  Set speed (1000.0 mm/s)
  MoveL 10131 to (504.54, 495.95, 18.9) mm, rotated rx 0 ry 90 rz 0 deg; joints [-11.552, -28.213, 111.281, -15.587, -82.457, 51.087]
  Set speed (1000.0 mm/s)
  MoveL 10132 to (501.11, 498.89, 18.9) mm, rotated rx 0 ry 90 rz 0 deg; joints [-11.886, -28.268, 111.619, -15.914, -82.741, 51.048]
  Set speed (30.0 mm/s)
  Call Extruder(0.111)
  MoveL 10133 to (503.8, 496.2, 18.9) mm, rotated rx 0 ry 90 rz 0 deg; joints [-11.588, -28.227, 111.363, -15.622, -82.525, 51.072]
  MoveL 10134 to (503.92, 496.08, 18.9) mm, rotated rx 0 ry 90 rz 0 deg; joints [-11.575, -28.225, 111.352, -15.608, -82.515, 51.073]
  Set speed (120.0 mm/s)
  MoveL 10135 to (504.54, 493.58, 18.9) mm, rotated rx 0 ry 90 rz 0 deg; joints [-11.335, -28.223, 111.338, -15.367, -82.497, 51.049]
  Set speed (1000.0 mm/s)
  MoveL 10136 to (495.89, 493.58, 18.9) mm, rotated rx 0 ry 90 rz 0 deg; joints [-11.496, -28.386, 112.372, -15.5, -83.341, 50.833]
  Set speed (1000.0 mm/s)
  MoveL 10137 to (498.94, 501.06, 18.9) mm, rotated rx 0 ry 90 rz 0 deg; joints [-12.126, -28.301, 111.823, -16.15, -82.913, 51.027]
  Set speed (30.0 mm/s)
  Call Extruder(0.126)
  MoveL 10138 to (495.87, 504.12, 18.9) mm, rotated rx 0 ry 90 rz 0 deg; joints [-12.469, -28.346, 112.108, -16.487, -83.155, 50.995]
  MoveL 10139 to (495.75, 504.25, 18.9) mm, rotated rx 0 ry 90 rz 0 deg; joints [-12.483, -28.347, 112.12, -16.501, -83.165, 50.994]
  Set speed (120.0 mm/s)
  MoveL 10140 to (495.98, 506.75, 18.9) mm, rotated rx 0 ry 90 rz 0 deg; joints [-12.708, -28.333, 112.027, -16.73, -83.096, 51.04]
  Set speed (1000.0 mm/s)
  MoveL 10141 to (504.36, 506.75, 18.9) mm, rotated rx 0 ry 90 rz 0 deg; joints [-12.537, -28.171, 111.026, -16.588, -82.287, 51.263]
  Set speed (1000.0 mm/s)
  MoveL 10142 to (503.43, 503.43, 18.9) mm, rotated rx 0 ry 90 rz 0 deg; joints [-12.254, -28.204, 111.225, -16.297, -82.436, 51.182]
  Set speed (30.0 mm/s)
  Call Extruder(0.243)
  MoveL 10143 to (509.32, 509.32, 18.9) mm, rotated rx 0 ry 90 rz 0 deg; joints [-12.669, -28.058, 110.36, -16.744, -81.762, 51.44]
  MoveL 10144 to (509.44, 509.44, 18.9) mm, rotated rx 0 ry 90 rz 0 deg; joints [-12.677, -28.055, 110.342, -16.753, -81.748, 51.445]
  Set speed (120.0 mm/s)
  MoveL 10145 to (495.98, 506.75, 18.9) mm, rotated rx 0 ry 90 rz 0 deg; joints [-12.708, -28.333, 112.027, -16.73, -83.096, 51.04]
  Set speed (1000.0 mm/s)
  MoveL 10146 to (495.94, 504.34, 18.9) mm, rotated rx 0 ry 90 rz 0 deg; joints [-12.487, -28.344, 112.096, -16.506, -83.145, 51]
  Set speed (1000.0 mm/s)
  MoveL 10147 to (496.01, 504.4, 18.9) mm, rotated rx 0 ry 90 rz 0 deg; joints [-12.492, -28.342, 112.085, -16.511, -83.137, 51.003]
  Set speed (15.0 mm/s)
  Call Extruder(0.067)
  MoveL 10148 to (496.01, 506.72, 18.9) mm, rotated rx 0 ry 90 rz 0 deg; joints [-12.705, -28.332, 112.024, -16.727, -83.094, 51.04]
  Call Extruder(0.242)
  MoveL 10149 to (504.33, 506.72, 18.9) mm, rotated rx 0 ry 90 rz 0 deg; joints [-12.535, -28.172, 111.03, -16.586, -82.29, 51.262]
  Call Extruder(0.027)
  MoveL 10150 to (504.33, 505.8, 18.9) mm, rotated rx 0 ry 90 rz 0 deg; joints [-12.452, -28.176, 111.055, -16.502, -82.307, 51.246]
  Call Extruder(0.306)
  MoveL 10151 to (499.53, 496.43, 18.9) mm, rotated rx 0 ry 90 rz 0 deg; joints [-11.69, -28.308, 111.869, -15.709, -82.937, 50.968]
  Call Extruder(0.017)
  MoveL 10152 to (499.27, 495.92, 18.9) mm, rotated rx 0 ry 90 rz 0 deg; joints [-11.648, -28.315, 111.913, -15.666, -82.971, 50.954]
  Call Extruder(0.010)
  MoveL 10153 to (499.84, 495.92, 18.9) mm, rotated rx 0 ry 90 rz 0 deg; joints [-11.637, -28.304, 111.844, -15.657, -82.916, 50.968]
  Call Extruder(0.000)
  MoveL 10154 to (499.84, 495.92, 18.9) mm, rotated rx 0 ry 90 rz 0 deg; joints [-11.637, -28.304, 111.844, -15.657, -82.915, 50.968]
  Call Extruder(0.136)
  MoveL 10155 to (504.51, 495.92, 18.9) mm, rotated rx 0 ry 90 rz 0 deg; joints [-11.55, -28.214, 111.285, -15.585, -82.461, 51.086]
  Call Extruder(0.067)
  MoveL 10156 to (504.51, 493.61, 18.9) mm, rotated rx 0 ry 90 rz 0 deg; joints [-11.338, -28.223, 111.341, -15.37, -82.499, 51.048]
  Call Extruder(0.250)
  MoveL 10157 to (495.92, 493.61, 18.9) mm, rotated rx 0 ry 90 rz 0 deg; joints [-11.498, -28.386, 112.368, -15.502, -83.338, 50.834]
  Call Extruder(0.027)
  MoveL 10158 to (495.92, 494.52, 18.9) mm, rotated rx 0 ry 90 rz 0 deg; joints [-11.583, -28.382, 112.346, -15.588, -83.322, 50.847]
  Call Extruder(0.306)
  MoveL 10159 to (500.7, 503.9, 18.9) mm, rotated rx 0 ry 90 rz 0 deg; joints [-12.351, -28.255, 111.539, -16.385, -82.691, 51.119]
  Call Extruder(0.017)
  MoveL 10160 to (500.96, 504.4, 18.9) mm, rotated rx 0 ry 90 rz 0 deg; joints [-12.392, -28.248, 111.494, -16.428, -82.657, 51.134]
  Call Extruder(0.010)
  MoveL 10161 to (500.39, 504.41, 18.9) mm, rotated rx 0 ry 90 rz 0 deg; joints [-12.404, -28.259, 111.562, -16.437, -82.712, 51.119]
  Call Extruder(0.000)
  MoveL 10162 to (500.39, 504.41, 18.9) mm, rotated rx 0 ry 90 rz 0 deg; joints [-12.404, -28.259, 111.563, -16.437, -82.712, 51.119]
  Call Extruder(0.128)
  MoveL 10163 to (496.01, 504.4, 18.9) mm, rotated rx 0 ry 90 rz 0 deg; joints [-12.492, -28.342, 112.085, -16.511, -83.137, 51.003]
  Set speed (120.0 mm/s)
  MoveL 10164 to (496.01, 504.8, 18.9) mm, rotated rx 0 ry 90 rz 0 deg; joints [-12.529, -28.34, 112.075, -16.548, -83.13, 51.01]
  Set speed (1000.0 mm/s)
  MoveL 10165 to (495.91, 504.81, 18.9) mm, rotated rx 0 ry 90 rz 0 deg; joints [-12.531, -28.342, 112.087, -16.55, -83.139, 51.007]
  Set speed (1000.0 mm/s)
  MoveL 10166 to (490.47, 509.53, 18.9) mm, rotated rx 0 ry 90 rz 0 deg; joints [-13.08, -28.421, 112.604, -17.088, -83.575, 50.935]
  Set speed (1000.0 mm/s)
  MoveL 10167 to (490.4, 509.6, 18.9) mm, rotated rx 0 ry 90 rz 0 deg; joints [-13.088, -28.422, 112.61, -17.095, -83.581, 50.934]
  Set speed (15.0 mm/s)
  Call Extruder(0.559)
  MoveL 10168 to (490.4, 490.4, 18.9) mm, rotated rx 0 ry 90 rz 0 deg; joints [-11.303, -28.495, 113.101, -15.288, -83.934, 50.648]
  MoveL 10169 to (509.6, 490.4, 18.9) mm, rotated rx 0 ry 90 rz 0 deg; joints [-10.955, -28.134, 110.804, -14.999, -82.055, 51.12]
  MoveL 10170 to (509.6, 509.6, 18.9) mm, rotated rx 0 ry 90 rz 0 deg; joints [-12.688, -28.051, 110.319, -16.765, -81.73, 51.452]
  MoveL 10171 to (490.4, 509.6, 18.9) mm, rotated rx 0 ry 90 rz 0 deg; joints [-13.088, -28.422, 112.61, -17.095, -83.581, 50.934]
  Set speed (120.0 mm/s)
  MoveL 10172 to (490.4, 509.2, 18.9) mm, rotated rx 0 ry 90 rz 0 deg; joints [-13.051, -28.424, 112.621, -17.058, -83.588, 50.928]
  Set speed (1000.0 mm/s)
  MoveL 10173 to (491.1, 508.9, 18.9) mm, rotated rx 0 ry 90 rz 0 deg; joints [-13.008, -28.413, 112.547, -17.017, -83.527, 50.942]
  Set speed (1000.0 mm/s)
  MoveL 10174 to (490.68, 490.68, 18.9) mm, rotated rx 0 ry 90 rz 0 deg; joints [-11.324, -28.489, 113.061, -15.31, -83.902, 50.659]
  Set speed (1000.0 mm/s)
  MoveL 10175 to (490.68, 490.68, 19) mm, rotated rx 0 ry 90 rz 0 deg; joints [-11.324, -28.5, 113.066, -15.31, -83.896, 50.661]
  Set speed (30.0 mm/s)
  Call Extruder(0.249)
  MoveL 10176 to (496.74, 496.74, 19) mm, rotated rx 0 ry 90 rz 0 deg; joints [-11.772, -28.37, 112.2, -15.783, -83.199, 50.903]
  MoveL 10177 to (496.86, 496.86, 19) mm, rotated rx 0 ry 90 rz 0 deg; joints [-11.781, -28.367, 112.182, -15.792, -83.185, 50.908]
  Set speed (120.0 mm/s)
  MoveL 10178 to (495.64, 494.46, 19) mm, rotated rx 0 ry 90 rz 0 deg; joints [-11.582, -28.398, 112.386, -15.587, -83.345, 50.841]
  Set speed (30.0 mm/s)
  Call Extruder(0.204)
  MoveL 10179 to (490.68, 499.42, 19) mm, rotated rx 0 ry 90 rz 0 deg; joints [-12.139, -28.468, 112.852, -16.135, -83.741, 50.787]
  Set speed (120.0 mm/s)
  MoveL 10180 to (490.68, 500.58, 19) mm, rotated rx 0 ry 90 rz 0 deg; joints [-12.247, -28.464, 112.822, -16.244, -83.72, 50.804]
  Set speed (30.0 mm/s)
  Call Extruder(0.208)
  MoveL 10181 to (495.73, 505.63, 19) mm, rotated rx 0 ry 90 rz 0 deg; joints [-12.61, -28.353, 112.091, -16.63, -83.136, 51.017]
  Set speed (120.0 mm/s)
  MoveL 10182 to (495.72, 504.27, 19) mm, rotated rx 0 ry 90 rz 0 deg; joints [-12.486, -28.358, 112.127, -16.504, -83.161, 50.995]
  Set speed (30.0 mm/s)
  Call Extruder(0.208)
  MoveL 10183 to (490.68, 509.32, 19) mm, rotated rx 0 ry 90 rz 0 deg; joints [-13.056, -28.429, 112.59, -17.064, -83.554, 50.939]
  MoveL 10184 to (490.56, 509.44, 19) mm, rotated rx 0 ry 90 rz 0 deg; joints [-13.07, -28.431, 112.601, -17.078, -83.563, 50.938]
  Set speed (120.0 mm/s)
  MoveL 10185 to (497.1, 507, 19) mm, rotated rx 0 ry 90 rz 0 deg; joints [-12.708, -28.322, 111.892, -16.734, -82.978, 51.076]
  Set speed (30.0 mm/s)
  Call Extruder(0.096)
  MoveL 10186 to (499.42, 509.32, 19) mm, rotated rx 0 ry 90 rz 0 deg; joints [-12.872, -28.267, 111.552, -16.909, -82.71, 51.177]
  Set speed (120.0 mm/s)
  MoveL 10187 to (500.58, 509.32, 19) mm, rotated rx 0 ry 90 rz 0 deg; joints [-12.847, -28.245, 111.414, -16.889, -82.599, 51.208]
  Set speed (30.0 mm/s)
  Call Extruder(0.096)
  MoveL 10188 to (502.9, 507, 19) mm, rotated rx 0 ry 90 rz 0 deg; joints [-12.589, -28.21, 111.199, -16.636, -82.417, 51.231]
  MoveL 10189 to (503.02, 506.87, 19) mm, rotated rx 0 ry 90 rz 0 deg; joints [-12.575, -28.208, 111.187, -16.622, -82.408, 51.232]
  Set speed (120.0 mm/s)
  MoveL 10190 to (504.46, 505.44, 19) mm, rotated rx 0 ry 90 rz 0 deg; joints [-12.416, -28.185, 111.054, -16.466, -82.295, 51.245]
  Set speed (30.0 mm/s)
  Call Extruder(0.200)
  MoveL 10191 to (509.32, 500.58, 19) mm, rotated rx 0 ry 90 rz 0 deg; joints [-11.882, -28.108, 110.594, -15.942, -81.91, 51.286]
  Set speed (120.0 mm/s)
  MoveL 10192 to (509.32, 499.42, 19) mm, rotated rx 0 ry 90 rz 0 deg; joints [-11.777, -28.113, 110.624, -15.835, -81.929, 51.266]
  Set speed (30.0 mm/s)
  Call Extruder(0.186)
  MoveL 10193 to (504.79, 494.89, 19) mm, rotated rx 0 ry 90 rz 0 deg; joints [-11.45, -28.223, 111.281, -15.485, -82.445, 51.077]
  Set speed (120.0 mm/s)
  MoveL 10194 to (504.79, 495.21, 19) mm, rotated rx 0 ry 90 rz 0 deg; joints [-11.479, -28.222, 111.274, -15.515, -82.44, 51.083]
  Set speed (30.0 mm/s)
  Call Extruder(0.186)
  MoveL 10195 to (509.32, 490.68, 19) mm, rotated rx 0 ry 90 rz 0 deg; joints [-10.985, -28.149, 110.836, -15.029, -82.072, 51.12]
  MoveL 10196 to (509.44, 490.56, 19) mm, rotated rx 0 ry 90 rz 0 deg; joints [-10.972, -28.147, 110.824, -15.016, -82.062, 51.121]
  Set speed (120.0 mm/s)
  MoveL 10197 to (503.23, 493.33, 19) mm, rotated rx 0 ry 90 rz 0 deg; joints [-11.336, -28.26, 111.507, -15.364, -82.624, 51.014]
  Set speed (30.0 mm/s)
  Call Extruder(0.109)
  MoveL 10198 to (500.58, 490.68, 19) mm, rotated rx 0 ry 90 rz 0 deg; joints [-11.141, -28.321, 111.887, -15.157, -82.926, 50.907]
  Set speed (120.0 mm/s)
  MoveL 10199 to (499.42, 490.68, 19) mm, rotated rx 0 ry 90 rz 0 deg; joints [-11.163, -28.343, 112.026, -15.174, -83.04, 50.878]
  Set speed (30.0 mm/s)
  MoveL 10200 to (496.77, 493.33, 19) mm, rotated rx 0 ry 90 rz 0 deg; joints [-11.456, -28.382, 112.279, -15.463, -83.254, 50.852]
  MoveL 10201 to (496.65, 493.45, 19) mm, rotated rx 0 ry 90 rz 0 deg; joints [-11.47, -28.384, 112.291, -15.476, -83.264, 50.851]
  Set speed (120.0 mm/s)
  MoveL 10202 to (504.54, 493.58, 19) mm, rotated rx 0 ry 90 rz 0 deg; joints [-11.335, -28.233, 111.343, -15.367, -82.492, 51.05]
  Set speed (1000.0 mm/s)
  MoveL 10203 to (504.54, 495.95, 19) mm, rotated rx 0 ry 90 rz 0 deg; joints [-11.552, -28.224, 111.286, -15.587, -82.452, 51.088]
  Set speed (1000.0 mm/s)
  MoveL 10204 to (501.11, 498.89, 19) mm, rotated rx 0 ry 90 rz 0 deg; joints [-11.886, -28.279, 111.624, -15.914, -82.736, 51.049]
  Set speed (30.0 mm/s)
  Call Extruder(0.111)
  MoveL 10205 to (503.8, 496.2, 19) mm, rotated rx 0 ry 90 rz 0 deg; joints [-11.588, -28.237, 111.368, -15.622, -82.52, 51.074]
  MoveL 10206 to (503.92, 496.08, 19) mm, rotated rx 0 ry 90 rz 0 deg; joints [-11.575, -28.236, 111.357, -15.609, -82.51, 51.075]
  Set speed (120.0 mm/s)
  MoveL 10207 to (504.54, 493.58, 19) mm, rotated rx 0 ry 90 rz 0 deg; joints [-11.335, -28.233, 111.343, -15.367, -82.492, 51.05]
  Set speed (1000.0 mm/s)
  MoveL 10208 to (495.89, 493.58, 19) mm, rotated rx 0 ry 90 rz 0 deg; joints [-11.496, -28.397, 112.378, -15.5, -83.336, 50.834]
  Set speed (1000.0 mm/s)
  MoveL 10209 to (498.94, 501.06, 19) mm, rotated rx 0 ry 90 rz 0 deg; joints [-12.126, -28.311, 111.828, -16.15, -82.908, 51.028]
  Set speed (30.0 mm/s)
  Call Extruder(0.126)
  MoveL 10210 to (495.87, 504.12, 19) mm, rotated rx 0 ry 90 rz 0 deg; joints [-12.469, -28.356, 112.114, -16.487, -83.15, 50.997]
  MoveL 10211 to (495.75, 504.25, 19) mm, rotated rx 0 ry 90 rz 0 deg; joints [-12.483, -28.358, 112.125, -16.501, -83.159, 50.995]
  Set speed (120.0 mm/s)
  MoveL 10212 to (495.98, 506.75, 19) mm, rotated rx 0 ry 90 rz 0 deg; joints [-12.708, -28.343, 112.032, -16.73, -83.091, 51.042]
  Set speed (1000.0 mm/s)
  MoveL 10213 to (504.36, 506.75, 19) mm, rotated rx 0 ry 90 rz 0 deg; joints [-12.537, -28.182, 111.031, -16.588, -82.282, 51.265]
  Set speed (1000.0 mm/s)
  MoveL 10214 to (503.43, 503.43, 19) mm, rotated rx 0 ry 90 rz 0 deg; joints [-12.254, -28.215, 111.23, -16.297, -82.431, 51.184]
  Set speed (30.0 mm/s)
  Call Extruder(0.243)
  MoveL 10215 to (509.32, 509.32, 19) mm, rotated rx 0 ry 90 rz 0 deg; joints [-12.669, -28.068, 110.365, -16.744, -81.757, 51.441]
  MoveL 10216 to (509.44, 509.44, 19) mm, rotated rx 0 ry 90 rz 0 deg; joints [-12.677, -28.065, 110.347, -16.753, -81.743, 51.447]
  Set speed (120.0 mm/s)
  MoveL 10217 to (495.98, 506.75, 19) mm, rotated rx 0 ry 90 rz 0 deg; joints [-12.708, -28.343, 112.032, -16.73, -83.091, 51.042]
  Set speed (1000.0 mm/s)
  MoveL 10218 to (495.94, 504.33, 19) mm, rotated rx 0 ry 90 rz 0 deg; joints [-12.487, -28.354, 112.101, -16.506, -83.14, 51.002]
  Set speed (1000.0 mm/s)
  MoveL 10219 to (496.01, 504.41, 19) mm, rotated rx 0 ry 90 rz 0 deg; joints [-12.492, -28.353, 112.09, -16.511, -83.132, 51.005]
  Set speed (15.0 mm/s)
  Call Extruder(0.067)
  MoveL 10220 to (496.01, 506.72, 19) mm, rotated rx 0 ry 90 rz 0 deg; joints [-12.705, -28.343, 112.029, -16.727, -83.089, 51.042]
  Call Extruder(0.242)
  MoveL 10221 to (504.33, 506.72, 19) mm, rotated rx 0 ry 90 rz 0 deg; joints [-12.535, -28.182, 111.035, -16.586, -82.285, 51.264]
  Call Extruder(0.027)
  MoveL 10222 to (504.33, 505.8, 19) mm, rotated rx 0 ry 90 rz 0 deg; joints [-12.452, -28.186, 111.06, -16.502, -82.301, 51.248]
  Call Extruder(0.306)
  MoveL 10223 to (499.53, 496.43, 19) mm, rotated rx 0 ry 90 rz 0 deg; joints [-11.69, -28.319, 111.874, -15.71, -82.932, 50.97]
  Call Extruder(0.017)
  MoveL 10224 to (499.27, 495.92, 19) mm, rotated rx 0 ry 90 rz 0 deg; joints [-11.648, -28.326, 111.918, -15.666, -82.966, 50.955]
  Call Extruder(0.010)
  MoveL 10225 to (499.84, 495.92, 19) mm, rotated rx 0 ry 90 rz 0 deg; joints [-11.637, -28.315, 111.849, -15.657, -82.91, 50.97]
  Call Extruder(0.000)
  MoveL 10226 to (499.84, 495.92, 19) mm, rotated rx 0 ry 90 rz 0 deg; joints [-11.637, -28.315, 111.849, -15.657, -82.91, 50.97]
  Call Extruder(0.136)
  MoveL 10227 to (504.51, 495.92, 19) mm, rotated rx 0 ry 90 rz 0 deg; joints [-11.55, -28.225, 111.29, -15.585, -82.455, 51.087]
  Call Extruder(0.067)
  MoveL 10228 to (504.51, 493.61, 19) mm, rotated rx 0 ry 90 rz 0 deg; joints [-11.338, -28.234, 111.346, -15.371, -82.494, 51.05]
  Call Extruder(0.250)
  MoveL 10229 to (495.92, 493.61, 19) mm, rotated rx 0 ry 90 rz 0 deg; joints [-11.498, -28.396, 112.373, -15.503, -83.332, 50.835]
  Call Extruder(0.027)
  MoveL 10230 to (495.92, 494.52, 19) mm, rotated rx 0 ry 90 rz 0 deg; joints [-11.583, -28.393, 112.351, -15.588, -83.317, 50.849]
  Call Extruder(0.306)
  MoveL 10231 to (500.7, 503.9, 19) mm, rotated rx 0 ry 90 rz 0 deg; joints [-12.351, -28.266, 111.544, -16.385, -82.686, 51.121]
  Call Extruder(0.017)
  MoveL 10232 to (500.96, 504.4, 19) mm, rotated rx 0 ry 90 rz 0 deg; joints [-12.392, -28.259, 111.499, -16.428, -82.652, 51.136]
  Call Extruder(0.010)
  MoveL 10233 to (500.39, 504.4, 19) mm, rotated rx 0 ry 90 rz 0 deg; joints [-12.404, -28.27, 111.568, -16.437, -82.707, 51.121]
  Call Extruder(0.000)
  MoveL 10234 to (500.39, 504.41, 19) mm, rotated rx 0 ry 90 rz 0 deg; joints [-12.404, -28.27, 111.568, -16.437, -82.707, 51.121]
  Call Extruder(0.128)
  MoveL 10235 to (496.01, 504.41, 19) mm, rotated rx 0 ry 90 rz 0 deg; joints [-12.492, -28.353, 112.09, -16.511, -83.132, 51.005]
  Set speed (120.0 mm/s)
  MoveL 10236 to (496.01, 504.81, 19) mm, rotated rx 0 ry 90 rz 0 deg; joints [-12.529, -28.351, 112.08, -16.548, -83.124, 51.011]
  Set speed (1000.0 mm/s)
  MoveL 10237 to (495.91, 504.8, 19) mm, rotated rx 0 ry 90 rz 0 deg; joints [-12.531, -28.353, 112.092, -16.55, -83.134, 51.008]
  Set speed (1000.0 mm/s)
  MoveL 10238 to (490.47, 509.53, 19) mm, rotated rx 0 ry 90 rz 0 deg; joints [-13.08, -28.432, 112.609, -17.088, -83.57, 50.937]
  Set speed (1000.0 mm/s)
  MoveL 10239 to (490.4, 509.6, 19) mm, rotated rx 0 ry 90 rz 0 deg; joints [-13.088, -28.433, 112.615, -17.096, -83.575, 50.936]
  Set speed (15.0 mm/s)
  Call Extruder(0.559)
  MoveL 10240 to (490.4, 490.4, 19) mm, rotated rx 0 ry 90 rz 0 deg; joints [-11.303, -28.505, 113.106, -15.288, -83.928, 50.65]
  MoveL 10241 to (509.6, 490.4, 19) mm, rotated rx 0 ry 90 rz 0 deg; joints [-10.955, -28.144, 110.809, -15, -82.049, 51.122]
  MoveL 10242 to (509.6, 509.6, 19) mm, rotated rx 0 ry 90 rz 0 deg; joints [-12.688, -28.061, 110.324, -16.765, -81.725, 51.454]
  MoveL 10243 to (490.4, 509.6, 19) mm, rotated rx 0 ry 90 rz 0 deg; joints [-13.088, -28.433, 112.615, -17.096, -83.575, 50.936]
  Set speed (120.0 mm/s)
  MoveL 10244 to (490.4, 509.2, 19) mm, rotated rx 0 ry 90 rz 0 deg; joints [-13.051, -28.435, 112.626, -17.058, -83.583, 50.929]
  Set speed (1000.0 mm/s)
  MoveL 10245 to (491.1, 508.9, 19) mm, rotated rx 0 ry 90 rz 0 deg; joints [-13.008, -28.423, 112.552, -17.017, -83.521, 50.944]
  Set speed (1000.0 mm/s)
  MoveL 10246 to (490.68, 490.68, 19) mm, rotated rx 0 ry 90 rz 0 deg; joints [-11.324, -28.5, 113.066, -15.31, -83.896, 50.661]
  Set speed (1000.0 mm/s)
  MoveL 10247 to (490.68, 490.68, 19.1) mm, rotated rx 0 ry 90 rz 0 deg; joints [-11.324, -28.51, 113.072, -15.31, -83.891, 50.662]
  Set speed (30.0 mm/s)
  Call Extruder(0.249)
  MoveL 10248 to (496.74, 496.74, 19.1) mm, rotated rx 0 ry 90 rz 0 deg; joints [-11.772, -28.38, 112.205, -15.783, -83.193, 50.905]
  MoveL 10249 to (496.86, 496.86, 19.1) mm, rotated rx 0 ry 90 rz 0 deg; joints [-11.781, -28.378, 112.187, -15.792, -83.179, 50.91]
  Set speed (120.0 mm/s)
  MoveL 10250 to (495.64, 494.46, 19.1) mm, rotated rx 0 ry 90 rz 0 deg; joints [-11.582, -28.409, 112.391, -15.587, -83.34, 50.842]
  Set speed (30.0 mm/s)
  Call Extruder(0.204)
  MoveL 10251 to (490.68, 499.42, 19.1) mm, rotated rx 0 ry 90 rz 0 deg; joints [-12.139, -28.479, 112.857, -16.135, -83.736, 50.788]
  Set speed (120.0 mm/s)
  MoveL 10252 to (490.68, 500.58, 19.1) mm, rotated rx 0 ry 90 rz 0 deg; joints [-12.247, -28.474, 112.827, -16.244, -83.714, 50.806]
  Set speed (30.0 mm/s)
  Call Extruder(0.208)
  MoveL 10253 to (495.73, 505.63, 19.1) mm, rotated rx 0 ry 90 rz 0 deg; joints [-12.61, -28.363, 112.097, -16.63, -83.131, 51.018]
  Set speed (120.0 mm/s)
  MoveL 10254 to (495.72, 504.27, 19.1) mm, rotated rx 0 ry 90 rz 0 deg; joints [-12.486, -28.369, 112.132, -16.504, -83.156, 50.997]
  Set speed (30.0 mm/s)
  Call Extruder(0.208)
  MoveL 10255 to (490.68, 509.32, 19.1) mm, rotated rx 0 ry 90 rz 0 deg; joints [-13.056, -28.44, 112.595, -17.064, -83.548, 50.941]
  MoveL 10256 to (490.56, 509.44, 19.1) mm, rotated rx 0 ry 90 rz 0 deg; joints [-13.07, -28.441, 112.606, -17.078, -83.558, 50.939]
  Set speed (120.0 mm/s)
  MoveL 10257 to (497.1, 507, 19.1) mm, rotated rx 0 ry 90 rz 0 deg; joints [-12.708, -28.332, 111.897, -16.734, -82.973, 51.078]
  Set speed (30.0 mm/s)
  Call Extruder(0.096)
  MoveL 10258 to (499.42, 509.32, 19.1) mm, rotated rx 0 ry 90 rz 0 deg; joints [-12.872, -28.278, 111.557, -16.91, -82.705, 51.179]
  Set speed (120.0 mm/s)
  MoveL 10259 to (500.58, 509.32, 19.1) mm, rotated rx 0 ry 90 rz 0 deg; joints [-12.847, -28.255, 111.419, -16.89, -82.593, 51.21]
  Set speed (30.0 mm/s)
  Call Extruder(0.096)
  MoveL 10260 to (502.9, 507, 19.1) mm, rotated rx 0 ry 90 rz 0 deg; joints [-12.589, -28.22, 111.204, -16.636, -82.412, 51.232]
  MoveL 10261 to (503.02, 506.87, 19.1) mm, rotated rx 0 ry 90 rz 0 deg; joints [-12.575, -28.218, 111.192, -16.622, -82.403, 51.233]
  Set speed (120.0 mm/s)
  MoveL 10262 to (504.46, 505.44, 19.1) mm, rotated rx 0 ry 90 rz 0 deg; joints [-12.416, -28.196, 111.059, -16.466, -82.29, 51.247]
  Set speed (30.0 mm/s)
  Call Extruder(0.200)
  MoveL 10263 to (509.32, 500.58, 19.1) mm, rotated rx 0 ry 90 rz 0 deg; joints [-11.882, -28.118, 110.599, -15.942, -81.905, 51.288]
  Set speed (120.0 mm/s)
  MoveL 10264 to (509.32, 499.42, 19.1) mm, rotated rx 0 ry 90 rz 0 deg; joints [-11.777, -28.123, 110.629, -15.835, -81.924, 51.268]
  Set speed (30.0 mm/s)
  Call Extruder(0.186)
  MoveL 10265 to (504.79, 494.89, 19.1) mm, rotated rx 0 ry 90 rz 0 deg; joints [-11.45, -28.234, 111.286, -15.486, -82.44, 51.079]
  Set speed (120.0 mm/s)
  MoveL 10266 to (504.79, 495.21, 19.1) mm, rotated rx 0 ry 90 rz 0 deg; joints [-11.479, -28.232, 111.279, -15.515, -82.435, 51.084]
  Set speed (30.0 mm/s)
  Call Extruder(0.186)
  MoveL 10267 to (509.32, 490.68, 19.1) mm, rotated rx 0 ry 90 rz 0 deg; joints [-10.985, -28.16, 110.841, -15.03, -82.067, 51.121]
  MoveL 10268 to (509.44, 490.56, 19.1) mm, rotated rx 0 ry 90 rz 0 deg; joints [-10.972, -28.158, 110.829, -15.017, -82.057, 51.122]
  Set speed (120.0 mm/s)
  MoveL 10269 to (503.23, 493.33, 19.1) mm, rotated rx 0 ry 90 rz 0 deg; joints [-11.336, -28.271, 111.512, -15.364, -82.619, 51.015]
  Set speed (30.0 mm/s)
  Call Extruder(0.109)
  MoveL 10270 to (500.58, 490.68, 19.1) mm, rotated rx 0 ry 90 rz 0 deg; joints [-11.141, -28.331, 111.892, -15.157, -82.921, 50.908]
  Set speed (120.0 mm/s)
  MoveL 10271 to (499.42, 490.68, 19.1) mm, rotated rx 0 ry 90 rz 0 deg; joints [-11.163, -28.353, 112.031, -15.174, -83.034, 50.88]
  Set speed (30.0 mm/s)
  MoveL 10272 to (496.77, 493.33, 19.1) mm, rotated rx 0 ry 90 rz 0 deg; joints [-11.456, -28.392, 112.284, -15.463, -83.249, 50.854]
  MoveL 10273 to (496.65, 493.45, 19.1) mm, rotated rx 0 ry 90 rz 0 deg; joints [-11.47, -28.394, 112.296, -15.477, -83.259, 50.853]
  Set speed (120.0 mm/s)
  MoveL 10274 to (504.54, 493.58, 19.1) mm, rotated rx 0 ry 90 rz 0 deg; joints [-11.335, -28.244, 111.348, -15.368, -82.486, 51.052]
  Set speed (1000.0 mm/s)
  MoveL 10275 to (504.54, 495.95, 19.1) mm, rotated rx 0 ry 90 rz 0 deg; joints [-11.552, -28.234, 111.291, -15.587, -82.447, 51.09]
  Set speed (1000.0 mm/s)
  MoveL 10276 to (501.11, 498.89, 19.1) mm, rotated rx 0 ry 90 rz 0 deg; joints [-11.886, -28.289, 111.629, -15.914, -82.73, 51.051]
  Set speed (30.0 mm/s)
  Call Extruder(0.111)
  MoveL 10277 to (503.8, 496.2, 19.1) mm, rotated rx 0 ry 90 rz 0 deg; joints [-11.588, -28.248, 111.374, -15.622, -82.515, 51.075]
  MoveL 10278 to (503.92, 496.08, 19.1) mm, rotated rx 0 ry 90 rz 0 deg; joints [-11.575, -28.246, 111.362, -15.609, -82.505, 51.076]
  Set speed (120.0 mm/s)
  MoveL 10279 to (504.54, 493.58, 19.1) mm, rotated rx 0 ry 90 rz 0 deg; joints [-11.335, -28.244, 111.348, -15.368, -82.486, 51.052]
  Set speed (1000.0 mm/s)
  MoveL 10280 to (495.89, 493.58, 19.1) mm, rotated rx 0 ry 90 rz 0 deg; joints [-11.496, -28.408, 112.383, -15.501, -83.33, 50.836]
  Set speed (1000.0 mm/s)
  MoveL 10281 to (498.94, 501.06, 19.1) mm, rotated rx 0 ry 90 rz 0 deg; joints [-12.126, -28.322, 111.833, -16.15, -82.903, 51.03]
  Set speed (30.0 mm/s)
  Call Extruder(0.126)
  MoveL 10282 to (495.87, 504.12, 19.1) mm, rotated rx 0 ry 90 rz 0 deg; joints [-12.469, -28.367, 112.119, -16.487, -83.144, 50.998]
  MoveL 10283 to (495.75, 504.25, 19.1) mm, rotated rx 0 ry 90 rz 0 deg; joints [-12.483, -28.369, 112.13, -16.501, -83.154, 50.997]
  Set speed (120.0 mm/s)
  MoveL 10284 to (495.98, 506.75, 19.1) mm, rotated rx 0 ry 90 rz 0 deg; joints [-12.708, -28.354, 112.037, -16.73, -83.085, 51.043]
  Set speed (1000.0 mm/s)
  MoveL 10285 to (504.36, 506.75, 19.1) mm, rotated rx 0 ry 90 rz 0 deg; joints [-12.537, -28.192, 111.036, -16.589, -82.276, 51.266]
  Set speed (1000.0 mm/s)
  MoveL 10286 to (503.43, 503.43, 19.1) mm, rotated rx 0 ry 90 rz 0 deg; joints [-12.254, -28.225, 111.235, -16.297, -82.426, 51.185]
  Set speed (30.0 mm/s)
  Call Extruder(0.243)
  MoveL 10287 to (509.32, 509.32, 19.1) mm, rotated rx 0 ry 90 rz 0 deg; joints [-12.669, -28.079, 110.37, -16.744, -81.752, 51.443]
  MoveL 10288 to (509.44, 509.44, 19.1) mm, rotated rx 0 ry 90 rz 0 deg; joints [-12.677, -28.076, 110.352, -16.753, -81.738, 51.448]
  Set speed (120.0 mm/s)
  MoveL 10289 to (495.98, 506.75, 19.1) mm, rotated rx 0 ry 90 rz 0 deg; joints [-12.708, -28.354, 112.037, -16.73, -83.085, 51.043]
  Set speed (1000.0 mm/s)
  MoveL 10290 to (495.94, 504.34, 19.1) mm, rotated rx 0 ry 90 rz 0 deg; joints [-12.487, -28.365, 112.106, -16.506, -83.134, 51.003]
  Set speed (1000.0 mm/s)
  MoveL 10291 to (496.01, 504.41, 19.1) mm, rotated rx 0 ry 90 rz 0 deg; joints [-12.492, -28.363, 112.096, -16.511, -83.126, 51.006]
  Set speed (15.0 mm/s)
  Call Extruder(0.067)
  MoveL 10292 to (496.01, 506.72, 19.1) mm, rotated rx 0 ry 90 rz 0 deg; joints [-12.705, -28.354, 112.034, -16.727, -83.083, 51.044]
  Call Extruder(0.242)
  MoveL 10293 to (504.33, 506.72, 19.1) mm, rotated rx 0 ry 90 rz 0 deg; joints [-12.535, -28.193, 111.04, -16.586, -82.28, 51.265]
  Call Extruder(0.027)
  MoveL 10294 to (504.33, 505.8, 19.1) mm, rotated rx 0 ry 90 rz 0 deg; joints [-12.452, -28.197, 111.065, -16.502, -82.296, 51.249]
  Call Extruder(0.306)
  MoveL 10295 to (499.53, 496.43, 19.1) mm, rotated rx 0 ry 90 rz 0 deg; joints [-11.69, -28.329, 111.879, -15.71, -82.926, 50.971]
  Call Extruder(0.017)
  MoveL 10296 to (499.27, 495.92, 19.1) mm, rotated rx 0 ry 90 rz 0 deg; joints [-11.648, -28.336, 111.923, -15.666, -82.961, 50.957]
  Call Extruder(0.010)
  MoveL 10297 to (499.84, 495.92, 19.1) mm, rotated rx 0 ry 90 rz 0 deg; joints [-11.637, -28.325, 111.854, -15.657, -82.905, 50.971]
  Call Extruder(0.000)
  MoveL 10298 to (499.84, 495.92, 19.1) mm, rotated rx 0 ry 90 rz 0 deg; joints [-11.637, -28.325, 111.854, -15.657, -82.905, 50.971]
  Call Extruder(0.136)
  MoveL 10299 to (504.51, 495.92, 19.1) mm, rotated rx 0 ry 90 rz 0 deg; joints [-11.55, -28.235, 111.295, -15.585, -82.45, 51.089]
  Call Extruder(0.067)
  MoveL 10300 to (504.51, 493.61, 19.1) mm, rotated rx 0 ry 90 rz 0 deg; joints [-11.338, -28.244, 111.351, -15.371, -82.489, 51.051]
  Call Extruder(0.250)
  MoveL 10301 to (495.92, 493.61, 19.1) mm, rotated rx 0 ry 90 rz 0 deg; joints [-11.498, -28.407, 112.379, -15.503, -83.327, 50.837]
  Call Extruder(0.027)
  MoveL 10302 to (495.92, 494.52, 19.1) mm, rotated rx 0 ry 90 rz 0 deg; joints [-11.583, -28.404, 112.356, -15.589, -83.311, 50.85]
  Call Extruder(0.306)
  MoveL 10303 to (500.7, 503.9, 19.1) mm, rotated rx 0 ry 90 rz 0 deg; joints [-12.351, -28.276, 111.549, -16.385, -82.681, 51.122]
  Call Extruder(0.017)
  MoveL 10304 to (500.96, 504.41, 19.1) mm, rotated rx 0 ry 90 rz 0 deg; joints [-12.392, -28.269, 111.504, -16.428, -82.646, 51.137]
  Call Extruder(0.010)
  MoveL 10305 to (500.39, 504.4, 19.1) mm, rotated rx 0 ry 90 rz 0 deg; joints [-12.404, -28.28, 111.573, -16.438, -82.702, 51.122]
  Call Extruder(0.000)
  MoveL 10306 to (500.39, 504.4, 19.1) mm, rotated rx 0 ry 90 rz 0 deg; joints [-12.404, -28.28, 111.573, -16.438, -82.702, 51.122]
  Call Extruder(0.128)
  MoveL 10307 to (496.01, 504.41, 19.1) mm, rotated rx 0 ry 90 rz 0 deg; joints [-12.492, -28.363, 112.096, -16.511, -83.126, 51.006]
  Set speed (120.0 mm/s)
  MoveL 10308 to (496.01, 504.81, 19.1) mm, rotated rx 0 ry 90 rz 0 deg; joints [-12.529, -28.362, 112.085, -16.549, -83.119, 51.013]
  Set speed (1000.0 mm/s)
  MoveL 10309 to (495.91, 504.8, 19.1) mm, rotated rx 0 ry 90 rz 0 deg; joints [-12.531, -28.363, 112.097, -16.55, -83.129, 51.01]
  Set speed (1000.0 mm/s)
  MoveL 10310 to (490.47, 509.53, 19.1) mm, rotated rx 0 ry 90 rz 0 deg; joints [-13.08, -28.443, 112.614, -17.088, -83.564, 50.938]
  Set speed (1000.0 mm/s)
  MoveL 10311 to (490.4, 509.6, 19.1) mm, rotated rx 0 ry 90 rz 0 deg; joints [-13.088, -28.444, 112.62, -17.096, -83.57, 50.937]
  Set speed (15.0 mm/s)
  Call Extruder(0.559)
  MoveL 10312 to (490.4, 490.4, 19.1) mm, rotated rx 0 ry 90 rz 0 deg; joints [-11.303, -28.516, 113.111, -15.288, -83.923, 50.651]
  MoveL 10313 to (509.6, 490.4, 19.1) mm, rotated rx 0 ry 90 rz 0 deg; joints [-10.955, -28.155, 110.814, -15, -82.044, 51.123]
  MoveL 10314 to (509.6, 509.6, 19.1) mm, rotated rx 0 ry 90 rz 0 deg; joints [-12.688, -28.072, 110.329, -16.765, -81.72, 51.456]
  MoveL 10315 to (490.4, 509.6, 19.1) mm, rotated rx 0 ry 90 rz 0 deg; joints [-13.088, -28.444, 112.62, -17.096, -83.57, 50.937]
  Set speed (120.0 mm/s)
  MoveL 10316 to (490.4, 509.2, 19.1) mm, rotated rx 0 ry 90 rz 0 deg; joints [-13.051, -28.445, 112.631, -17.058, -83.578, 50.931]
  Set speed (1000.0 mm/s)
  MoveL 10317 to (491.1, 508.9, 19.1) mm, rotated rx 0 ry 90 rz 0 deg; joints [-13.008, -28.434, 112.557, -17.018, -83.516, 50.946]
  Set speed (1000.0 mm/s)
  MoveL 10318 to (490.68, 490.68, 19.1) mm, rotated rx 0 ry 90 rz 0 deg; joints [-11.324, -28.51, 113.072, -15.31, -83.891, 50.662]
  Set speed (1000.0 mm/s)
  MoveL 10319 to (490.68, 490.68, 19.2) mm, rotated rx 0 ry 90 rz 0 deg; joints [-11.324, -28.521, 113.077, -15.31, -83.885, 50.664]
  Set speed (30.0 mm/s)
  Call Extruder(0.249)
  MoveL 10320 to (496.74, 496.74, 19.2) mm, rotated rx 0 ry 90 rz 0 deg; joints [-11.772, -28.391, 112.21, -15.783, -83.188, 50.906]
  MoveL 10321 to (496.86, 496.86, 19.2) mm, rotated rx 0 ry 90 rz 0 deg; joints [-11.781, -28.388, 112.192, -15.793, -83.174, 50.911]
  Set speed (120.0 mm/s)
  MoveL 10322 to (495.64, 494.46, 19.2) mm, rotated rx 0 ry 90 rz 0 deg; joints [-11.582, -28.42, 112.397, -15.587, -83.335, 50.844]
  Set speed (30.0 mm/s)
  Call Extruder(0.204)
  MoveL 10323 to (490.68, 499.42, 19.2) mm, rotated rx 0 ry 90 rz 0 deg; joints [-12.139, -28.489, 112.862, -16.135, -83.73, 50.79]
  Set speed (120.0 mm/s)
  MoveL 10324 to (490.68, 500.58, 19.2) mm, rotated rx 0 ry 90 rz 0 deg; joints [-12.247, -28.485, 112.832, -16.244, -83.709, 50.807]
  Set speed (30.0 mm/s)
  Call Extruder(0.208)
  MoveL 10325 to (495.73, 505.63, 19.2) mm, rotated rx 0 ry 90 rz 0 deg; joints [-12.61, -28.374, 112.102, -16.63, -83.126, 51.02]
  Set speed (120.0 mm/s)
  MoveL 10326 to (495.72, 504.27, 19.2) mm, rotated rx 0 ry 90 rz 0 deg; joints [-12.486, -28.38, 112.137, -16.504, -83.151, 50.998]
  Set speed (30.0 mm/s)
  Call Extruder(0.208)
  MoveL 10327 to (490.68, 509.32, 19.2) mm, rotated rx 0 ry 90 rz 0 deg; joints [-13.056, -28.45, 112.6, -17.065, -83.543, 50.942]
  MoveL 10328 to (490.56, 509.44, 19.2) mm, rotated rx 0 ry 90 rz 0 deg; joints [-13.07, -28.452, 112.611, -17.078, -83.553, 50.941]
  Set speed (120.0 mm/s)
  MoveL 10329 to (497.1, 507, 19.2) mm, rotated rx 0 ry 90 rz 0 deg; joints [-12.708, -28.343, 111.902, -16.734, -82.967, 51.079]
  Set speed (30.0 mm/s)
  Call Extruder(0.096)
  MoveL 10330 to (499.42, 509.32, 19.2) mm, rotated rx 0 ry 90 rz 0 deg; joints [-12.872, -28.288, 111.562, -16.91, -82.7, 51.18]
  Set speed (120.0 mm/s)
  MoveL 10331 to (500.58, 509.32, 19.2) mm, rotated rx 0 ry 90 rz 0 deg; joints [-12.847, -28.266, 111.424, -16.89, -82.588, 51.212]
  Set speed (30.0 mm/s)
  Call Extruder(0.096)
  MoveL 10332 to (502.9, 507, 19.2) mm, rotated rx 0 ry 90 rz 0 deg; joints [-12.589, -28.231, 111.209, -16.636, -82.407, 51.234]
  MoveL 10333 to (503.02, 506.87, 19.2) mm, rotated rx 0 ry 90 rz 0 deg; joints [-12.575, -28.229, 111.197, -16.623, -82.397, 51.235]
  Set speed (120.0 mm/s)
  MoveL 10334 to (504.46, 505.44, 19.2) mm, rotated rx 0 ry 90 rz 0 deg; joints [-12.416, -28.207, 111.064, -16.467, -82.285, 51.248]
  Set speed (30.0 mm/s)
  Call Extruder(0.200)
  MoveL 10335 to (509.32, 500.58, 19.2) mm, rotated rx 0 ry 90 rz 0 deg; joints [-11.882, -28.129, 110.604, -15.942, -81.899, 51.289]
  Set speed (120.0 mm/s)
  MoveL 10336 to (509.32, 499.42, 19.2) mm, rotated rx 0 ry 90 rz 0 deg; joints [-11.777, -28.134, 110.634, -15.836, -81.919, 51.269]
  Set speed (30.0 mm/s)
  Call Extruder(0.186)
  MoveL 10337 to (504.79, 494.89, 19.2) mm, rotated rx 0 ry 90 rz 0 deg; joints [-11.45, -28.244, 111.291, -15.486, -82.435, 51.08]
  Set speed (120.0 mm/s)
  MoveL 10338 to (504.79, 495.21, 19.2) mm, rotated rx 0 ry 90 rz 0 deg; joints [-11.479, -28.243, 111.284, -15.515, -82.429, 51.086]
  Set speed (30.0 mm/s)
  Call Extruder(0.186)
  MoveL 10339 to (509.32, 490.68, 19.2) mm, rotated rx 0 ry 90 rz 0 deg; joints [-10.985, -28.17, 110.846, -15.03, -82.062, 51.123]
  MoveL 10340 to (509.44, 490.56, 19.2) mm, rotated rx 0 ry 90 rz 0 deg; joints [-10.972, -28.168, 110.834, -15.017, -82.052, 51.124]
  Set speed (120.0 mm/s)
  MoveL 10341 to (503.23, 493.33, 19.2) mm, rotated rx 0 ry 90 rz 0 deg; joints [-11.336, -28.281, 111.517, -15.364, -82.613, 51.016]
  Set speed (30.0 mm/s)
  Call Extruder(0.109)
  MoveL 10342 to (500.58, 490.68, 19.2) mm, rotated rx 0 ry 90 rz 0 deg; joints [-11.141, -28.342, 111.898, -15.157, -82.916, 50.91]
  Set speed (120.0 mm/s)
  MoveL 10343 to (499.42, 490.68, 19.2) mm, rotated rx 0 ry 90 rz 0 deg; joints [-11.163, -28.364, 112.036, -15.175, -83.029, 50.881]
  Set speed (30.0 mm/s)
  MoveL 10344 to (496.77, 493.33, 19.2) mm, rotated rx 0 ry 90 rz 0 deg; joints [-11.456, -28.403, 112.289, -15.463, -83.243, 50.855]
  MoveL 10345 to (496.65, 493.45, 19.2) mm, rotated rx 0 ry 90 rz 0 deg; joints [-11.47, -28.405, 112.301, -15.477, -83.253, 50.854]
  Set speed (120.0 mm/s)
  MoveL 10346 to (504.54, 493.58, 19.2) mm, rotated rx 0 ry 90 rz 0 deg; joints [-11.335, -28.254, 111.353, -15.368, -82.481, 51.053]
  Set speed (1000.0 mm/s)
  MoveL 10347 to (504.54, 495.95, 19.2) mm, rotated rx 0 ry 90 rz 0 deg; joints [-11.552, -28.245, 111.296, -15.588, -82.441, 51.091]
  Set speed (1000.0 mm/s)
  MoveL 10348 to (501.11, 498.89, 19.2) mm, rotated rx 0 ry 90 rz 0 deg; joints [-11.886, -28.3, 111.634, -15.914, -82.725, 51.052]
  Set speed (30.0 mm/s)
  Call Extruder(0.111)
  MoveL 10349 to (503.8, 496.2, 19.2) mm, rotated rx 0 ry 90 rz 0 deg; joints [-11.588, -28.259, 111.379, -15.622, -82.509, 51.077]
  MoveL 10350 to (503.92, 496.08, 19.2) mm, rotated rx 0 ry 90 rz 0 deg; joints [-11.575, -28.257, 111.367, -15.609, -82.5, 51.078]
  Set speed (120.0 mm/s)
  MoveL 10351 to (504.54, 493.58, 19.2) mm, rotated rx 0 ry 90 rz 0 deg; joints [-11.335, -28.254, 111.353, -15.368, -82.481, 51.053]
  Set speed (1000.0 mm/s)
  MoveL 10352 to (495.89, 493.58, 19.2) mm, rotated rx 0 ry 90 rz 0 deg; joints [-11.496, -28.418, 112.388, -15.501, -83.325, 50.837]
  Set speed (1000.0 mm/s)
  MoveL 10353 to (498.94, 501.06, 19.2) mm, rotated rx 0 ry 90 rz 0 deg; joints [-12.126, -28.333, 111.838, -16.151, -82.897, 51.031]
  Set speed (30.0 mm/s)
  Call Extruder(0.126)
  MoveL 10354 to (495.87, 504.12, 19.2) mm, rotated rx 0 ry 90 rz 0 deg; joints [-12.469, -28.377, 112.124, -16.488, -83.139, 51]
  MoveL 10355 to (495.75, 504.25, 19.2) mm, rotated rx 0 ry 90 rz 0 deg; joints [-12.483, -28.379, 112.135, -16.501, -83.149, 50.999]
  Set speed (120.0 mm/s)
  MoveL 10356 to (495.98, 506.75, 19.2) mm, rotated rx 0 ry 90 rz 0 deg; joints [-12.708, -28.365, 112.042, -16.73, -83.08, 51.045]
  Set speed (1000.0 mm/s)
  MoveL 10357 to (504.35, 506.75, 19.2) mm, rotated rx 0 ry 90 rz 0 deg; joints [-12.537, -28.203, 111.041, -16.589, -82.271, 51.268]
  Set speed (1000.0 mm/s)
  MoveL 10358 to (503.43, 503.43, 19.2) mm, rotated rx 0 ry 90 rz 0 deg; joints [-12.254, -28.236, 111.24, -16.297, -82.42, 51.187]
  Set speed (30.0 mm/s)
  Call Extruder(0.243)
  MoveL 10359 to (509.32, 509.32, 19.2) mm, rotated rx 0 ry 90 rz 0 deg; joints [-12.669, -28.089, 110.375, -16.744, -81.746, 51.445]
  MoveL 10360 to (509.44, 509.44, 19.2) mm, rotated rx 0 ry 90 rz 0 deg; joints [-12.677, -28.086, 110.357, -16.753, -81.732, 51.45]
  Set speed (120.0 mm/s)
  MoveL 10361 to (495.98, 506.75, 19.2) mm, rotated rx 0 ry 90 rz 0 deg; joints [-12.708, -28.365, 112.042, -16.73, -83.08, 51.045]
  Set speed (1000.0 mm/s)
  MoveL 10362 to (495.94, 504.34, 19.2) mm, rotated rx 0 ry 90 rz 0 deg; joints [-12.487, -28.375, 112.111, -16.506, -83.129, 51.005]
  Set speed (1000.0 mm/s)
  MoveL 10363 to (496.01, 504.41, 19.2) mm, rotated rx 0 ry 90 rz 0 deg; joints [-12.492, -28.374, 112.101, -16.512, -83.121, 51.008]
  Set speed (15.0 mm/s)
  Call Extruder(0.067)
  MoveL 10364 to (496.01, 506.72, 19.2) mm, rotated rx 0 ry 90 rz 0 deg; joints [-12.705, -28.364, 112.039, -16.727, -83.078, 51.045]
  Call Extruder(0.242)
  MoveL 10365 to (504.33, 506.72, 19.2) mm, rotated rx 0 ry 90 rz 0 deg; joints [-12.535, -28.203, 111.045, -16.587, -82.274, 51.267]
  Call Extruder(0.027)
  MoveL 10366 to (504.33, 505.8, 19.2) mm, rotated rx 0 ry 90 rz 0 deg; joints [-12.452, -28.208, 111.07, -16.502, -82.291, 51.251]
  Call Extruder(0.306)
  MoveL 10367 to (499.53, 496.43, 19.2) mm, rotated rx 0 ry 90 rz 0 deg; joints [-11.69, -28.34, 111.884, -15.71, -82.921, 50.973]
  Call Extruder(0.017)
  MoveL 10368 to (499.27, 495.92, 19.2) mm, rotated rx 0 ry 90 rz 0 deg; joints [-11.648, -28.347, 111.928, -15.667, -82.955, 50.958]
  Call Extruder(0.010)
  MoveL 10369 to (499.84, 495.92, 19.2) mm, rotated rx 0 ry 90 rz 0 deg; joints [-11.637, -28.336, 111.86, -15.658, -82.9, 50.973]
  Call Extruder(0.000)
  MoveL 10370 to (499.84, 495.92, 19.2) mm, rotated rx 0 ry 90 rz 0 deg; joints [-11.637, -28.336, 111.859, -15.658, -82.899, 50.973]
  Call Extruder(0.136)
  MoveL 10371 to (504.51, 495.92, 19.2) mm, rotated rx 0 ry 90 rz 0 deg; joints [-11.55, -28.246, 111.3, -15.585, -82.445, 51.09]
  Call Extruder(0.067)
  MoveL 10372 to (504.51, 493.61, 19.2) mm, rotated rx 0 ry 90 rz 0 deg; joints [-11.338, -28.255, 111.356, -15.371, -82.483, 51.053]
  Call Extruder(0.250)
  MoveL 10373 to (495.92, 493.61, 19.2) mm, rotated rx 0 ry 90 rz 0 deg; joints [-11.498, -28.418, 112.384, -15.503, -83.322, 50.838]
  Call Extruder(0.027)
  MoveL 10374 to (495.92, 494.52, 19.2) mm, rotated rx 0 ry 90 rz 0 deg; joints [-11.583, -28.414, 112.361, -15.589, -83.306, 50.852]
  Call Extruder(0.306)
  MoveL 10375 to (500.7, 503.9, 19.2) mm, rotated rx 0 ry 90 rz 0 deg; joints [-12.351, -28.287, 111.554, -16.385, -82.675, 51.124]
  Call Extruder(0.017)
  MoveL 10376 to (500.96, 504.4, 19.2) mm, rotated rx 0 ry 90 rz 0 deg; joints [-12.392, -28.28, 111.509, -16.428, -82.641, 51.139]
  Call Extruder(0.010)
  MoveL 10377 to (500.39, 504.4, 19.2) mm, rotated rx 0 ry 90 rz 0 deg; joints [-12.404, -28.291, 111.578, -16.438, -82.696, 51.124]
  Call Extruder(0.000)
  MoveL 10378 to (500.39, 504.41, 19.2) mm, rotated rx 0 ry 90 rz 0 deg; joints [-12.404, -28.291, 111.578, -16.438, -82.696, 51.124]
  Call Extruder(0.128)
  MoveL 10379 to (496.01, 504.41, 19.2) mm, rotated rx 0 ry 90 rz 0 deg; joints [-12.492, -28.374, 112.101, -16.512, -83.121, 51.008]
  Set speed (120.0 mm/s)
  MoveL 10380 to (496.01, 504.81, 19.2) mm, rotated rx 0 ry 90 rz 0 deg; joints [-12.529, -28.372, 112.09, -16.549, -83.114, 51.014]
  Set speed (1000.0 mm/s)
  MoveL 10381 to (495.91, 504.81, 19.2) mm, rotated rx 0 ry 90 rz 0 deg; joints [-12.531, -28.374, 112.102, -16.551, -83.123, 51.012]
  Set speed (1000.0 mm/s)
  MoveL 10382 to (490.47, 509.53, 19.2) mm, rotated rx 0 ry 90 rz 0 deg; joints [-13.08, -28.453, 112.619, -17.088, -83.559, 50.94]
  Set speed (1000.0 mm/s)
  MoveL 10383 to (490.4, 509.6, 19.2) mm, rotated rx 0 ry 90 rz 0 deg; joints [-13.088, -28.454, 112.625, -17.096, -83.565, 50.939]
  Set speed (15.0 mm/s)
  Call Extruder(0.559)
  MoveL 10384 to (490.4, 490.4, 19.2) mm, rotated rx 0 ry 90 rz 0 deg; joints [-11.303, -28.527, 113.116, -15.288, -83.918, 50.653]
  MoveL 10385 to (509.6, 490.4, 19.2) mm, rotated rx 0 ry 90 rz 0 deg; joints [-10.955, -28.165, 110.819, -15, -82.039, 51.125]
  MoveL 10386 to (509.6, 509.6, 19.2) mm, rotated rx 0 ry 90 rz 0 deg; joints [-12.688, -28.082, 110.334, -16.765, -81.714, 51.457]
  MoveL 10387 to (490.4, 509.6, 19.2) mm, rotated rx 0 ry 90 rz 0 deg; joints [-13.088, -28.454, 112.625, -17.096, -83.565, 50.939]
  Set speed (120.0 mm/s)
  MoveL 10388 to (490.4, 509.2, 19.2) mm, rotated rx 0 ry 90 rz 0 deg; joints [-13.051, -28.456, 112.636, -17.059, -83.572, 50.933]
  Set speed (1000.0 mm/s)
  MoveL 10389 to (491.1, 508.9, 19.2) mm, rotated rx 0 ry 90 rz 0 deg; joints [-13.008, -28.445, 112.562, -17.018, -83.511, 50.947]
  Set speed (1000.0 mm/s)
  MoveL 10390 to (490.4, 509.6, 19.2) mm, rotated rx 0 ry 90 rz 0 deg; joints [-13.088, -28.454, 112.625, -17.096, -83.565, 50.939]
  Set speed (1000.0 mm/s)
  MoveL 10391 to (490.4, 509.6, 19.3) mm, rotated rx 0 ry 90 rz 0 deg; joints [-13.088, -28.465, 112.63, -17.096, -83.559, 50.941]
  Set speed (15.0 mm/s)
  MoveL 10392 to (490.4, 490.4, 19.3) mm, rotated rx 0 ry 90 rz 0 deg; joints [-11.303, -28.537, 113.121, -15.289, -83.912, 50.654]
  MoveL 10393 to (509.6, 490.4, 19.3) mm, rotated rx 0 ry 90 rz 0 deg; joints [-10.955, -28.176, 110.824, -15, -82.033, 51.126]
  MoveL 10394 to (509.6, 509.6, 19.3) mm, rotated rx 0 ry 90 rz 0 deg; joints [-12.688, -28.093, 110.339, -16.766, -81.709, 51.459]
  MoveL 10395 to (490.4, 509.6, 19.3) mm, rotated rx 0 ry 90 rz 0 deg; joints [-13.088, -28.465, 112.63, -17.096, -83.559, 50.941]
  Set speed (120.0 mm/s)
  MoveL 10396 to (490.4, 509.2, 19.3) mm, rotated rx 0 ry 90 rz 0 deg; joints [-13.051, -28.467, 112.641, -17.059, -83.567, 50.934]
  Set speed (1000.0 mm/s)
  MoveL 10397 to (490.5, 509.2, 19.3) mm, rotated rx 0 ry 90 rz 0 deg; joints [-13.049, -28.465, 112.629, -17.057, -83.557, 50.937]
  Set speed (1000.0 mm/s)
  MoveL 10398 to (495.94, 504.33, 19.3) mm, rotated rx 0 ry 90 rz 0 deg; joints [-12.487, -28.386, 112.116, -16.506, -83.124, 51.006]
  Set speed (1000.0 mm/s)
  MoveL 10399 to (496.01, 504.41, 19.3) mm, rotated rx 0 ry 90 rz 0 deg; joints [-12.492, -28.384, 112.106, -16.512, -83.116, 51.009]
  Set speed (15.0 mm/s)
  Call Extruder(0.067)
  MoveL 10400 to (496.01, 506.72, 19.3) mm, rotated rx 0 ry 90 rz 0 deg; joints [-12.705, -28.375, 112.044, -16.727, -83.073, 51.047]
  Call Extruder(0.242)
  MoveL 10401 to (504.33, 506.72, 19.3) mm, rotated rx 0 ry 90 rz 0 deg; joints [-12.535, -28.214, 111.05, -16.587, -82.269, 51.268]
  Call Extruder(0.027)
  MoveL 10402 to (504.33, 505.8, 19.3) mm, rotated rx 0 ry 90 rz 0 deg; joints [-12.452, -28.218, 111.075, -16.502, -82.286, 51.253]
  Call Extruder(0.306)
  MoveL 10403 to (499.53, 496.43, 19.3) mm, rotated rx 0 ry 90 rz 0 deg; joints [-11.69, -28.35, 111.889, -15.71, -82.916, 50.974]
  Call Extruder(0.017)
  MoveL 10404 to (499.27, 495.92, 19.3) mm, rotated rx 0 ry 90 rz 0 deg; joints [-11.648, -28.357, 111.933, -15.667, -82.95, 50.96]
  Call Extruder(0.010)
  MoveL 10405 to (499.84, 495.92, 19.3) mm, rotated rx 0 ry 90 rz 0 deg; joints [-11.637, -28.347, 111.865, -15.658, -82.894, 50.974]
  Call Extruder(0.000)
  MoveL 10406 to (499.84, 495.92, 19.3) mm, rotated rx 0 ry 90 rz 0 deg; joints [-11.637, -28.347, 111.864, -15.658, -82.894, 50.974]
  Call Extruder(0.136)
  MoveL 10407 to (504.51, 495.92, 19.3) mm, rotated rx 0 ry 90 rz 0 deg; joints [-11.55, -28.256, 111.305, -15.586, -82.439, 51.092]
  Call Extruder(0.067)
  MoveL 10408 to (504.51, 493.61, 19.3) mm, rotated rx 0 ry 90 rz 0 deg; joints [-11.338, -28.265, 111.361, -15.371, -82.478, 51.054]
  Call Extruder(0.250)
  MoveL 10409 to (495.92, 493.61, 19.3) mm, rotated rx 0 ry 90 rz 0 deg; joints [-11.498, -28.428, 112.389, -15.503, -83.316, 50.84]
  Call Extruder(0.027)
  MoveL 10410 to (495.92, 494.52, 19.3) mm, rotated rx 0 ry 90 rz 0 deg; joints [-11.583, -28.425, 112.366, -15.589, -83.301, 50.853]
  Call Extruder(0.306)
  MoveL 10411 to (500.7, 503.9, 19.3) mm, rotated rx 0 ry 90 rz 0 deg; joints [-12.351, -28.298, 111.559, -16.386, -82.67, 51.125]
  Call Extruder(0.017)
  MoveL 10412 to (500.96, 504.41, 19.3) mm, rotated rx 0 ry 90 rz 0 deg; joints [-12.392, -28.29, 111.514, -16.429, -82.636, 51.14]
  Call Extruder(0.010)
  MoveL 10413 to (500.39, 504.4, 19.3) mm, rotated rx 0 ry 90 rz 0 deg; joints [-12.404, -28.301, 111.583, -16.438, -82.691, 51.125]
  Call Extruder(0.000)
  MoveL 10414 to (500.39, 504.4, 19.3) mm, rotated rx 0 ry 90 rz 0 deg; joints [-12.404, -28.301, 111.583, -16.438, -82.691, 51.125]
  Call Extruder(0.128)
  MoveL 10415 to (496.01, 504.41, 19.3) mm, rotated rx 0 ry 90 rz 0 deg; joints [-12.492, -28.384, 112.106, -16.512, -83.116, 51.009]
  Set speed (120.0 mm/s)
  MoveL 10416 to (496.01, 504.81, 19.3) mm, rotated rx 0 ry 90 rz 0 deg; joints [-12.529, -28.383, 112.095, -16.549, -83.108, 51.016]
  Set speed (1000.0 mm/s)
  MoveL 10417 to (495.91, 504.8, 19.3) mm, rotated rx 0 ry 90 rz 0 deg; joints [-12.531, -28.385, 112.107, -16.551, -83.118, 51.013]
  Set speed (1000.0 mm/s)
  MoveL 10418 to (495.32, 503.71, 19.3) mm, rotated rx 0 ry 90 rz 0 deg; joints [-12.443, -28.4, 112.206, -16.459, -83.195, 50.98]
  Set speed (15.0 mm/s)
  Call Extruder(0.107)
  MoveL 10419 to (495.32, 507.41, 19.3) mm, rotated rx 0 ry 90 rz 0 deg; joints [-12.782, -28.385, 112.108, -16.804, -83.126, 51.04]
  Call Extruder(0.282)
  MoveL 10420 to (505.02, 507.41, 19.3) mm, rotated rx 0 ry 90 rz 0 deg; joints [-12.583, -28.197, 110.949, -16.639, -82.19, 51.299]
  Call Extruder(0.052)
  MoveL 10421 to (505.02, 505.64, 19.3) mm, rotated rx 0 ry 90 rz 0 deg; joints [-12.423, -28.205, 110.996, -16.476, -82.222, 51.268]
  Call Extruder(0.295)
  MoveL 10422 to (500.4, 496.61, 19.3) mm, rotated rx 0 ry 90 rz 0 deg; joints [-11.69, -28.333, 111.781, -15.713, -82.828, 50.999]
  Call Extruder(0.140)
  MoveL 10423 to (505.2, 496.61, 19.3) mm, rotated rx 0 ry 90 rz 0 deg; joints [-11.6, -28.24, 111.205, -15.639, -82.361, 51.12]
  Call Extruder(0.107)
  MoveL 10424 to (505.2, 492.92, 19.3) mm, rotated rx 0 ry 90 rz 0 deg; joints [-11.263, -28.254, 111.295, -15.297, -82.422, 51.06]
  Call Extruder(0.290)
  MoveL 10425 to (495.23, 492.92, 19.3) mm, rotated rx 0 ry 90 rz 0 deg; joints [-11.447, -28.443, 112.487, -15.449, -83.396, 50.812]
  Call Extruder(0.052)
  MoveL 10426 to (495.23, 494.69, 19.3) mm, rotated rx 0 ry 90 rz 0 deg; joints [-11.611, -28.437, 112.444, -15.616, -83.365, 50.838]
  Call Extruder(0.295)
  MoveL 10427 to (499.84, 503.72, 19.3) mm, rotated rx 0 ry 90 rz 0 deg; joints [-12.352, -28.315, 111.667, -16.383, -82.757, 51.099]
  Call Extruder(0.132)
  MoveL 10428 to (495.32, 503.71, 19.3) mm, rotated rx 0 ry 90 rz 0 deg; joints [-12.443, -28.4, 112.206, -16.459, -83.195, 50.98]
  Set speed (120.0 mm/s)
  MoveL 10429 to (491.09, 508.91, 19.3) mm, rotated rx 0 ry 90 rz 0 deg; joints [-13.01, -28.455, 112.568, -17.019, -83.506, 50.949]
  Set speed (15.0 mm/s)
  Call Extruder(0.519)
  MoveL 10430 to (491.09, 491.09, 19.3) mm, rotated rx 0 ry 90 rz 0 deg; joints [-11.355, -28.523, 113.023, -15.343, -83.833, 50.681]
  MoveL 10431 to (508.91, 491.09, 19.3) mm, rotated rx 0 ry 90 rz 0 deg; joints [-11.03, -28.187, 110.891, -15.074, -82.09, 51.121]
  MoveL 10432 to (508.91, 508.91, 19.3) mm, rotated rx 0 ry 90 rz 0 deg; joints [-12.64, -28.11, 110.44, -16.714, -81.788, 51.428]
  MoveL 10433 to (491.09, 508.91, 19.3) mm, rotated rx 0 ry 90 rz 0 deg; joints [-13.01, -28.455, 112.568, -17.019, -83.506, 50.949]
  Set speed (120.0 mm/s)
  MoveL 10434 to (491.77, 508.59, 19.3) mm, rotated rx 0 ry 90 rz 0 deg; joints [-12.966, -28.445, 112.496, -16.977, -83.447, 50.962]
  Set speed (15.0 mm/s)
  Call Extruder(0.015)
  MoveL 10435 to (491.4, 508.23, 19.3) mm, rotated rx 0 ry 90 rz 0 deg; joints [-12.94, -28.453, 112.549, -16.95, -83.489, 50.947]
  Set speed (120.0 mm/s)
  MoveL 10436 to (491.4, 507.24, 19.3) mm, rotated rx 0 ry 90 rz 0 deg; joints [-12.849, -28.457, 112.576, -16.857, -83.508, 50.931]
  Set speed (15.0 mm/s)
  Call Extruder(0.056)
  MoveL 10437 to (492.76, 508.59, 19.3) mm, rotated rx 0 ry 90 rz 0 deg; joints [-12.945, -28.427, 112.379, -16.96, -83.351, 50.989]
  Set speed (120.0 mm/s)
  MoveL 10438 to (493.75, 508.59, 19.3) mm, rotated rx 0 ry 90 rz 0 deg; joints [-12.924, -28.409, 112.262, -16.942, -83.256, 51.016]
  Set speed (15.0 mm/s)
  Call Extruder(0.096)
  MoveL 10439 to (491.4, 506.25, 19.3) mm, rotated rx 0 ry 90 rz 0 deg; joints [-12.758, -28.461, 112.602, -16.765, -83.527, 50.915]
  Set speed (120.0 mm/s)
  MoveL 10440 to (491.4, 505.26, 19.3) mm, rotated rx 0 ry 90 rz 0 deg; joints [-12.666, -28.465, 112.629, -16.672, -83.546, 50.9]
  Set speed (15.0 mm/s)
  Call Extruder(0.137)
  MoveL 10441 to (494.74, 508.59, 19.3) mm, rotated rx 0 ry 90 rz 0 deg; joints [-12.903, -28.391, 112.144, -16.924, -83.16, 51.043]
  Set speed (120.0 mm/s)
  MoveL 10442 to (495.72, 508.59, 19.3) mm, rotated rx 0 ry 90 rz 0 deg; joints [-12.882, -28.372, 112.027, -16.907, -83.065, 51.07]
  Set speed (15.0 mm/s)
  Call Extruder(0.178)
  MoveL 10443 to (491.4, 504.27, 19.3) mm, rotated rx 0 ry 90 rz 0 deg; joints [-12.574, -28.469, 112.655, -16.579, -83.564, 50.884]
  Set speed (120.0 mm/s)
  MoveL 10444 to (491.4, 503.28, 19.3) mm, rotated rx 0 ry 90 rz 0 deg; joints [-12.483, -28.473, 112.681, -16.486, -83.583, 50.869]
  Set speed (15.0 mm/s)
  Call Extruder(0.148)
  MoveL 10445 to (495, 506.88, 19.3) mm, rotated rx 0 ry 90 rz 0 deg; joints [-12.74, -28.393, 112.159, -16.76, -83.167, 51.023]
  Set speed (120.0 mm/s)
  MoveL 10446 to (495, 505.89, 19.3) mm, rotated rx 0 ry 90 rz 0 deg; joints [-12.649, -28.397, 112.186, -16.668, -83.185, 51.007]
  Set speed (15.0 mm/s)
  Call Extruder(0.148)
  MoveL 10447 to (491.4, 502.29, 19.3) mm, rotated rx 0 ry 90 rz 0 deg; joints [-12.391, -28.476, 112.707, -16.393, -83.601, 50.854]
  Set speed (120.0 mm/s)
  MoveL 10448 to (491.4, 501.3, 19.3) mm, rotated rx 0 ry 90 rz 0 deg; joints [-12.299, -28.48, 112.733, -16.3, -83.62, 50.839]
  Set speed (15.0 mm/s)
  MoveL 10449 to (495, 504.9, 19.3) mm, rotated rx 0 ry 90 rz 0 deg; joints [-12.558, -28.401, 112.212, -16.575, -83.204, 50.991]
  Set speed (120.0 mm/s)
  MoveL 10450 to (495, 503.91, 19.3) mm, rotated rx 0 ry 90 rz 0 deg; joints [-12.467, -28.405, 112.238, -16.483, -83.222, 50.975]
  Set speed (15.0 mm/s)
  MoveL 10451 to (491.4, 500.31, 19.3) mm, rotated rx 0 ry 90 rz 0 deg; joints [-12.208, -28.484, 112.758, -16.207, -83.638, 50.824]
  Set speed (120.0 mm/s)
  MoveL 10452 to (491.4, 499.32, 19.3) mm, rotated rx 0 ry 90 rz 0 deg; joints [-12.116, -28.488, 112.783, -16.114, -83.656, 50.809]
  Set speed (15.0 mm/s)
  Call Extruder(0.168)
  MoveL 10453 to (495.48, 503.4, 19.3) mm, rotated rx 0 ry 90 rz 0 deg; joints [-12.41, -28.398, 112.195, -16.427, -83.185, 50.979]
  Set speed (120.0 mm/s)
  MoveL 10454 to (496.47, 503.4, 19.3) mm, rotated rx 0 ry 90 rz 0 deg; joints [-12.39, -28.38, 112.077, -16.41, -83.089, 51.006]
  Set speed (15.0 mm/s)
  Call Extruder(0.208)
  MoveL 10455 to (491.4, 498.33, 19.3) mm, rotated rx 0 ry 90 rz 0 deg; joints [-12.024, -28.492, 112.808, -16.021, -83.674, 50.794]
  Set speed (120.0 mm/s)
  MoveL 10456 to (491.4, 497.34, 19.3) mm, rotated rx 0 ry 90 rz 0 deg; joints [-11.932, -28.495, 112.833, -15.928, -83.692, 50.78]
  Set speed (15.0 mm/s)
  Call Extruder(0.249)
  MoveL 10457 to (497.46, 503.4, 19.3) mm, rotated rx 0 ry 90 rz 0 deg; joints [-12.37, -28.361, 111.959, -16.393, -82.993, 51.032]
  Set speed (120.0 mm/s)
  MoveL 10458 to (498.45, 503.4, 19.3) mm, rotated rx 0 ry 90 rz 0 deg; joints [-12.351, -28.343, 111.841, -16.377, -82.897, 51.058]
  Set speed (15.0 mm/s)
  Call Extruder(0.290)
  MoveL 10459 to (491.4, 496.35, 19.3) mm, rotated rx 0 ry 90 rz 0 deg; joints [-11.839, -28.499, 112.858, -15.834, -83.71, 50.765]
  Set speed (120.0 mm/s)
  MoveL 10460 to (491.4, 495.36, 19.3) mm, rotated rx 0 ry 90 rz 0 deg; joints [-11.747, -28.502, 112.882, -15.741, -83.727, 50.751]
  Set speed (15.0 mm/s)
  Call Extruder(0.321)
  MoveL 10461 to (499.2, 503.16, 19.3) mm, rotated rx 0 ry 90 rz 0 deg; joints [-12.313, -28.33, 111.758, -16.342, -82.829, 51.073]
  MoveL 10462 to (499.32, 503.28, 19.3) mm, rotated rx 0 ry 90 rz 0 deg; joints [-12.322, -28.327, 111.74, -16.351, -82.815, 51.079]
  Set speed (120.0 mm/s)
  MoveL 10463 to (498.17, 501.14, 19.3) mm, rotated rx 0 ry 90 rz 0 deg; joints [-12.149, -28.357, 111.933, -16.171, -82.966, 51.014]
  Set speed (15.0 mm/s)
  Call Extruder(0.278)
  MoveL 10464 to (491.4, 494.37, 19.3) mm, rotated rx 0 ry 90 rz 0 deg; joints [-11.655, -28.506, 112.907, -15.648, -83.745, 50.736]
  Set speed (120.0 mm/s)
  MoveL 10465 to (491.4, 493.38, 19.3) mm, rotated rx 0 ry 90 rz 0 deg; joints [-11.563, -28.51, 112.931, -15.554, -83.762, 50.722]
  Set speed (15.0 mm/s)
  Call Extruder(0.236)
  MoveL 10466 to (497.13, 499.12, 19.3) mm, rotated rx 0 ry 90 rz 0 deg; joints [-11.983, -28.385, 112.108, -15.999, -83.102, 50.955]
  MoveL 10467 to (497.26, 499.24, 19.3) mm, rotated rx 0 ry 90 rz 0 deg; joints [-11.992, -28.382, 112.09, -16.009, -83.088, 50.96]
  Set speed (120.0 mm/s)
  MoveL 10468 to (496.1, 497.09, 19.3) mm, rotated rx 0 ry 90 rz 0 deg; joints [-11.817, -28.412, 112.281, -15.827, -83.238, 50.897]
  Set speed (15.0 mm/s)
  Call Extruder(0.193)
  MoveL 10469 to (491.4, 492.39, 19.3) mm, rotated rx 0 ry 90 rz 0 deg; joints [-11.47, -28.513, 112.955, -15.461, -83.779, 50.708]
  Set speed (120.0 mm/s)
  MoveL 10470 to (491.4, 491.4, 19.3) mm, rotated rx 0 ry 90 rz 0 deg; joints [-11.378, -28.517, 112.979, -15.367, -83.796, 50.694]
  Set speed (15.0 mm/s)
  Call Extruder(0.151)
  MoveL 10471 to (495.07, 495.07, 19.3) mm, rotated rx 0 ry 90 rz 0 deg; joints [-11.65, -28.438, 112.454, -15.654, -83.374, 50.84]
  Set speed (120.0 mm/s)
  MoveL 10472 to (494.92, 493.93, 19.3) mm, rotated rx 0 ry 90 rz 0 deg; joints [-11.546, -28.445, 112.501, -15.549, -83.409, 50.819]
  Set speed (15.0 mm/s)
  Call Extruder(0.104)
  MoveL 10473 to (492.39, 491.4, 19.3) mm, rotated rx 0 ry 90 rz 0 deg; joints [-11.36, -28.499, 112.861, -15.352, -83.699, 50.719]
  Set speed (120.0 mm/s)
  MoveL 10474 to (493.38, 491.4, 19.3) mm, rotated rx 0 ry 90 rz 0 deg; joints [-11.341, -28.482, 112.744, -15.336, -83.602, 50.743]
  Set speed (15.0 mm/s)
  Call Extruder(0.063)
  MoveL 10475 to (494.92, 492.94, 19.3) mm, rotated rx 0 ry 90 rz 0 deg; joints [-11.455, -28.449, 112.525, -15.456, -83.426, 50.804]
  Set speed (120.0 mm/s)
  MoveL 10476 to (495.57, 492.6, 19.3) mm, rotated rx 0 ry 90 rz 0 deg; joints [-11.411, -28.438, 112.455, -15.414, -83.368, 50.816]
  Set speed (15.0 mm/s)
  Call Extruder(0.049)
  MoveL 10477 to (494.37, 491.4, 19.3) mm, rotated rx 0 ry 90 rz 0 deg; joints [-11.323, -28.464, 112.626, -15.32, -83.505, 50.768]
  Set speed (120.0 mm/s)
  MoveL 10478 to (495.36, 491.4, 19.3) mm, rotated rx 0 ry 90 rz 0 deg; joints [-11.304, -28.446, 112.508, -15.305, -83.408, 50.793]
  Set speed (15.0 mm/s)
  MoveL 10479 to (496.56, 492.6, 19.3) mm, rotated rx 0 ry 90 rz 0 deg; joints [-11.393, -28.42, 112.337, -15.399, -83.271, 50.841]
  Set speed (120.0 mm/s)
  MoveL 10480 to (497.55, 492.6, 19.3) mm, rotated rx 0 ry 90 rz 0 deg; joints [-11.374, -28.402, 112.219, -15.383, -83.174, 50.866]
  Set speed (15.0 mm/s)
  MoveL 10481 to (496.35, 491.4, 19.3) mm, rotated rx 0 ry 90 rz 0 deg; joints [-11.286, -28.428, 112.39, -15.29, -83.312, 50.818]
  Set speed (120.0 mm/s)
  MoveL 10482 to (497.34, 491.4, 19.3) mm, rotated rx 0 ry 90 rz 0 deg; joints [-11.268, -28.41, 112.272, -15.274, -83.215, 50.842]
  Set speed (15.0 mm/s)
  MoveL 10483 to (498.54, 492.6, 19.3) mm, rotated rx 0 ry 90 rz 0 deg; joints [-11.356, -28.384, 112.101, -15.368, -83.077, 50.89]
  Set speed (120.0 mm/s)
  MoveL 10484 to (499.53, 492.6, 19.3) mm, rotated rx 0 ry 90 rz 0 deg; joints [-11.338, -28.365, 111.982, -15.353, -82.981, 50.915]
  Set speed (15.0 mm/s)
  MoveL 10485 to (498.33, 491.4, 19.3) mm, rotated rx 0 ry 90 rz 0 deg; joints [-11.249, -28.392, 112.154, -15.259, -83.118, 50.867]
  Set speed (120.0 mm/s)
  MoveL 10486 to (499.32, 491.4, 19.3) mm, rotated rx 0 ry 90 rz 0 deg; joints [-11.231, -28.374, 112.036, -15.244, -83.021, 50.891]
  Set speed (15.0 mm/s)
  MoveL 10487 to (500.52, 492.6, 19.3) mm, rotated rx 0 ry 90 rz 0 deg; joints [-11.319, -28.346, 111.864, -15.338, -82.884, 50.939]
  Set speed (120.0 mm/s)
  MoveL 10488 to (501.51, 492.6, 19.3) mm, rotated rx 0 ry 90 rz 0 deg; joints [-11.301, -28.328, 111.745, -15.323, -82.787, 50.964]
  Set speed (15.0 mm/s)
  MoveL 10489 to (500.31, 491.4, 19.3) mm, rotated rx 0 ry 90 rz 0 deg; joints [-11.213, -28.355, 111.917, -15.229, -82.924, 50.916]
  Set speed (120.0 mm/s)
  MoveL 10490 to (501.3, 491.4, 19.3) mm, rotated rx 0 ry 90 rz 0 deg; joints [-11.195, -28.336, 111.799, -15.214, -82.827, 50.94]
  Set speed (15.0 mm/s)
  MoveL 10491 to (502.5, 492.6, 19.3) mm, rotated rx 0 ry 90 rz 0 deg; joints [-11.283, -28.309, 111.627, -15.308, -82.691, 50.989]
  Set speed (120.0 mm/s)
  MoveL 10492 to (503.49, 492.6, 19.3) mm, rotated rx 0 ry 90 rz 0 deg; joints [-11.265, -28.289, 111.508, -15.293, -82.594, 51.013]
  Set speed (15.0 mm/s)
  MoveL 10493 to (502.29, 491.4, 19.3) mm, rotated rx 0 ry 90 rz 0 deg; joints [-11.177, -28.317, 111.68, -15.199, -82.731, 50.965]
  Set speed (120.0 mm/s)
  MoveL 10494 to (503.28, 491.4, 19.3) mm, rotated rx 0 ry 90 rz 0 deg; joints [-11.159, -28.298, 111.561, -15.185, -82.634, 50.989]
  Set speed (15.0 mm/s)
  Call Extruder(0.049)
  MoveL 10495 to (504.48, 492.6, 19.3) mm, rotated rx 0 ry 90 rz 0 deg; joints [-11.247, -28.27, 111.389, -15.278, -82.497, 51.037]
  Set speed (120.0 mm/s)
  MoveL 10496 to (505.47, 492.6, 19.3) mm, rotated rx 0 ry 90 rz 0 deg; joints [-11.229, -28.25, 111.27, -15.264, -82.401, 51.062]
  Set speed (15.0 mm/s)
  MoveL 10497 to (504.27, 491.4, 19.3) mm, rotated rx 0 ry 90 rz 0 deg; joints [-11.141, -28.279, 111.442, -15.17, -82.537, 51.013]
  Set speed (120.0 mm/s)
  MoveL 10498 to (505.26, 491.4, 19.3) mm, rotated rx 0 ry 90 rz 0 deg; joints [-11.123, -28.259, 111.323, -15.156, -82.441, 51.037]
  Set speed (15.0 mm/s)
  Call Extruder(0.137)
  MoveL 10499 to (508.59, 494.74, 19.3) mm, rotated rx 0 ry 90 rz 0 deg; joints [-11.366, -28.179, 110.842, -15.415, -82.062, 51.173]
  Set speed (120.0 mm/s)
  MoveL 10500 to (508.59, 495.72, 19.3) mm, rotated rx 0 ry 90 rz 0 deg; joints [-11.456, -28.175, 110.818, -15.506, -82.046, 51.19]
  Set speed (15.0 mm/s)
  Call Extruder(0.127)
  MoveL 10501 to (505.52, 492.65, 19.3) mm, rotated rx 0 ry 90 rz 0 deg; joints [-11.232, -28.249, 111.263, -15.267, -82.396, 51.064]
  Set speed (120.0 mm/s)
  MoveL 10502 to (505.52, 493.64, 19.3) mm, rotated rx 0 ry 90 rz 0 deg; joints [-11.323, -28.245, 111.24, -15.359, -82.38, 51.079]
  Set speed (15.0 mm/s)
  MoveL 10503 to (508.59, 496.71, 19.3) mm, rotated rx 0 ry 90 rz 0 deg; joints [-11.546, -28.171, 110.794, -15.598, -82.029, 51.207]
  Set speed (120.0 mm/s)
  MoveL 10504 to (508.59, 497.7, 19.3) mm, rotated rx 0 ry 90 rz 0 deg; joints [-11.636, -28.167, 110.769, -15.689, -82.013, 51.223]
  Set speed (15.0 mm/s)
  MoveL 10505 to (505.52, 494.63, 19.3) mm, rotated rx 0 ry 90 rz 0 deg; joints [-11.413, -28.241, 111.216, -15.451, -82.363, 51.096]
  Set speed (120.0 mm/s)
  MoveL 10506 to (505.52, 495.62, 19.3) mm, rotated rx 0 ry 90 rz 0 deg; joints [-11.503, -28.237, 111.191, -15.542, -82.347, 51.112]
  Set speed (15.0 mm/s)
  MoveL 10507 to (508.59, 498.69, 19.3) mm, rotated rx 0 ry 90 rz 0 deg; joints [-11.725, -28.162, 110.744, -15.78, -81.996, 51.24]
  Set speed (120.0 mm/s)
  MoveL 10508 to (508.59, 499.68, 19.3) mm, rotated rx 0 ry 90 rz 0 deg; joints [-11.815, -28.158, 110.72, -15.871, -81.979, 51.257]
  Set speed (15.0 mm/s)
  MoveL 10509 to (505.52, 496.61, 19.3) mm, rotated rx 0 ry 90 rz 0 deg; joints [-11.593, -28.233, 111.167, -15.634, -82.33, 51.128]
  Set speed (120.0 mm/s)
  MoveL 10510 to (504.84, 496.93, 19.3) mm, rotated rx 0 ry 90 rz 0 deg; joints [-11.635, -28.245, 111.24, -15.674, -82.39, 51.116]
  Set speed (15.0 mm/s)
  Call Extruder(0.154)
  MoveL 10511 to (508.59, 500.67, 19.3) mm, rotated rx 0 ry 90 rz 0 deg; joints [-11.904, -28.154, 110.695, -15.962, -81.963, 51.274]
  Set speed (120.0 mm/s)
  MoveL 10512 to (508.59, 501.66, 19.3) mm, rotated rx 0 ry 90 rz 0 deg; joints [-11.994, -28.15, 110.669, -16.053, -81.946, 51.291]
  Set speed (15.0 mm/s)
  Call Extruder(0.195)
  MoveL 10513 to (503.86, 496.93, 19.3) mm, rotated rx 0 ry 90 rz 0 deg; joints [-11.654, -28.265, 111.359, -15.689, -82.486, 51.092]
  Set speed (120.0 mm/s)
  MoveL 10514 to (502.86, 496.93, 19.3) mm, rotated rx 0 ry 90 rz 0 deg; joints [-11.672, -28.284, 111.478, -15.704, -82.583, 51.067]
  Set speed (15.0 mm/s)
  Call Extruder(0.236)
  MoveL 10515 to (508.59, 502.65, 19.3) mm, rotated rx 0 ry 90 rz 0 deg; joints [-12.083, -28.145, 110.644, -16.144, -81.929, 51.309]
  Set speed (120.0 mm/s)
  MoveL 10516 to (508.59, 503.64, 19.3) mm, rotated rx 0 ry 90 rz 0 deg; joints [-12.172, -28.141, 110.618, -16.235, -81.912, 51.326]
  Set speed (15.0 mm/s)
  Call Extruder(0.277)
  MoveL 10517 to (501.87, 496.93, 19.3) mm, rotated rx 0 ry 90 rz 0 deg; joints [-11.691, -28.304, 111.596, -15.72, -82.679, 51.042]
  Set speed (120.0 mm/s)
  MoveL 10518 to (500.94, 496.98, 19.3) mm, rotated rx 0 ry 90 rz 0 deg; joints [-11.714, -28.321, 111.707, -15.739, -82.769, 51.019]
  Set speed (15.0 mm/s)
  Call Extruder(0.315)
  MoveL 10519 to (508.59, 504.63, 19.3) mm, rotated rx 0 ry 90 rz 0 deg; joints [-12.262, -28.136, 110.592, -16.326, -81.894, 51.343]
  Set speed (120.0 mm/s)
  MoveL 10520 to (508.59, 505.62, 19.3) mm, rotated rx 0 ry 90 rz 0 deg; joints [-12.351, -28.132, 110.566, -16.417, -81.877, 51.361]
  Set speed (15.0 mm/s)
  Call Extruder(0.272)
  MoveL 10521 to (501.98, 499.01, 19.3) mm, rotated rx 0 ry 90 rz 0 deg; joints [-11.879, -28.293, 111.532, -15.911, -82.633, 51.078]
  MoveL 10522 to (501.85, 498.88, 19.3) mm, rotated rx 0 ry 90 rz 0 deg; joints [-11.871, -28.296, 111.55, -15.902, -82.647, 51.073]
  Set speed (120.0 mm/s)
  MoveL 10523 to (503.02, 501.04, 19.3) mm, rotated rx 0 ry 90 rz 0 deg; joints [-12.044, -28.265, 111.356, -16.083, -82.497, 51.138]
  Set speed (15.0 mm/s)
  Call Extruder(0.230)
  MoveL 10524 to (508.59, 506.61, 19.3) mm, rotated rx 0 ry 90 rz 0 deg; joints [-12.44, -28.127, 110.54, -16.508, -81.859, 51.378]
  Set speed (120.0 mm/s)
  MoveL 10525 to (508.59, 507.6, 19.3) mm, rotated rx 0 ry 90 rz 0 deg; joints [-12.529, -28.123, 110.514, -16.599, -81.842, 51.396]
  Set speed (15.0 mm/s)
  Call Extruder(0.187)
  MoveL 10526 to (504.05, 503.06, 19.3) mm, rotated rx 0 ry 90 rz 0 deg; joints [-12.209, -28.235, 111.179, -16.254, -82.361, 51.199]
  MoveL 10527 to (503.93, 502.94, 19.3) mm, rotated rx 0 ry 90 rz 0 deg; joints [-12.2, -28.238, 111.197, -16.245, -82.375, 51.193]
  Set speed (120.0 mm/s)
  MoveL 10528 to (505.09, 505.09, 19.3) mm, rotated rx 0 ry 90 rz 0 deg; joints [-12.372, -28.206, 111.002, -16.425, -82.224, 51.26]
  Set speed (15.0 mm/s)
  Call Extruder(0.144)
  MoveL 10529 to (508.59, 508.59, 19.3) mm, rotated rx 0 ry 90 rz 0 deg; joints [-12.618, -28.118, 110.487, -16.69, -81.824, 51.414]
  Set speed (120.0 mm/s)
  MoveL 10530 to (507.6, 508.59, 19.3) mm, rotated rx 0 ry 90 rz 0 deg; joints [-12.638, -28.139, 110.606, -16.706, -81.919, 51.388]
  Set speed (15.0 mm/s)
  Call Extruder(0.094)
  MoveL 10531 to (505.33, 506.32, 19.3) mm, rotated rx 0 ry 90 rz 0 deg; joints [-12.479, -28.196, 110.94, -16.534, -82.179, 51.288]
  Set speed (120.0 mm/s)
  MoveL 10532 to (505.33, 507.31, 19.3) mm, rotated rx 0 ry 90 rz 0 deg; joints [-12.568, -28.191, 110.914, -16.625, -82.161, 51.305]
  Set speed (15.0 mm/s)
  Call Extruder(0.053)
  MoveL 10533 to (506.61, 508.59, 19.3) mm, rotated rx 0 ry 90 rz 0 deg; joints [-12.658, -28.159, 110.725, -16.722, -82.015, 51.362]
  Set speed (120.0 mm/s)
  MoveL 10534 to (505.62, 508.59, 19.3) mm, rotated rx 0 ry 90 rz 0 deg; joints [-12.678, -28.179, 110.844, -16.738, -82.11, 51.335]
  Set speed (15.0 mm/s)
  Call Extruder(0.036)
  MoveL 10535 to (504.75, 507.72, 19.3) mm, rotated rx 0 ry 90 rz 0 deg; joints [-12.617, -28.201, 110.972, -16.672, -82.21, 51.297]
  Set speed (120.0 mm/s)
  MoveL 10536 to (504.63, 508.59, 19.3) mm, rotated rx 0 ry 90 rz 0 deg; joints [-12.698, -28.199, 110.963, -16.755, -82.205, 51.309]
  Set speed (15.0 mm/s)
  MoveL 10537 to (503.76, 507.72, 19.3) mm, rotated rx 0 ry 90 rz 0 deg; joints [-12.637, -28.221, 111.091, -16.689, -82.305, 51.271]
  Set speed (120.0 mm/s)
  MoveL 10538 to (503.64, 508.59, 19.3) mm, rotated rx 0 ry 90 rz 0 deg; joints [-12.719, -28.219, 111.082, -16.771, -82.301, 51.283]
  Set speed (15.0 mm/s)
  MoveL 10539 to (502.77, 507.72, 19.3) mm, rotated rx 0 ry 90 rz 0 deg; joints [-12.657, -28.24, 111.21, -16.705, -82.401, 51.245]
  Set speed (120.0 mm/s)
  MoveL 10540 to (502.65, 508.59, 19.3) mm, rotated rx 0 ry 90 rz 0 deg; joints [-12.739, -28.239, 111.2, -16.788, -82.396, 51.256]
  Set speed (15.0 mm/s)
  MoveL 10541 to (501.78, 507.72, 19.3) mm, rotated rx 0 ry 90 rz 0 deg; joints [-12.678, -28.26, 111.328, -16.722, -82.496, 51.218]
  Set speed (120.0 mm/s)
  MoveL 10542 to (501.66, 508.59, 19.3) mm, rotated rx 0 ry 90 rz 0 deg; joints [-12.759, -28.258, 111.319, -16.805, -82.492, 51.23]
  Set speed (15.0 mm/s)
  MoveL 10543 to (500.79, 507.72, 19.3) mm, rotated rx 0 ry 90 rz 0 deg; joints [-12.698, -28.279, 111.447, -16.739, -82.592, 51.192]
  Set speed (120.0 mm/s)
  MoveL 10544 to (500.67, 508.59, 19.3) mm, rotated rx 0 ry 90 rz 0 deg; joints [-12.78, -28.278, 111.437, -16.821, -82.587, 51.203]
  Set speed (15.0 mm/s)
  MoveL 10545 to (499.8, 507.72, 19.3) mm, rotated rx 0 ry 90 rz 0 deg; joints [-12.718, -28.299, 111.565, -16.755, -82.687, 51.165]
  Set speed (120.0 mm/s)
  MoveL 10546 to (499.68, 508.59, 19.3) mm, rotated rx 0 ry 90 rz 0 deg; joints [-12.8, -28.297, 111.555, -16.838, -82.682, 51.177]
  Set speed (15.0 mm/s)
  MoveL 10547 to (498.81, 507.72, 19.3) mm, rotated rx 0 ry 90 rz 0 deg; joints [-12.739, -28.318, 111.683, -16.772, -82.783, 51.139]
  Set speed (120.0 mm/s)
  MoveL 10548 to (498.69, 508.59, 19.3) mm, rotated rx 0 ry 90 rz 0 deg; joints [-12.821, -28.316, 111.674, -16.855, -82.778, 51.15]
  Set speed (15.0 mm/s)
  MoveL 10549 to (497.82, 507.72, 19.3) mm, rotated rx 0 ry 90 rz 0 deg; joints [-12.759, -28.336, 111.801, -16.789, -82.878, 51.112]
  Set speed (120.0 mm/s)
  MoveL 10550 to (497.7, 508.59, 19.3) mm, rotated rx 0 ry 90 rz 0 deg; joints [-12.841, -28.335, 111.791, -16.872, -82.873, 51.124]
  Set speed (15.0 mm/s)
  Call Extruder(0.036)
  MoveL 10551 to (496.83, 507.72, 19.3) mm, rotated rx 0 ry 90 rz 0 deg; joints [-12.779, -28.355, 111.919, -16.806, -82.974, 51.086]
  Set speed (120.0 mm/s)
  MoveL 10552 to (496.71, 508.59, 19.3) mm, rotated rx 0 ry 90 rz 0 deg; joints [-12.862, -28.354, 111.909, -16.89, -82.969, 51.097]
  Set speed (15.0 mm/s)
  MoveL 10553 to (495.84, 507.72, 19.3) mm, rotated rx 0 ry 90 rz 0 deg; joints [-12.8, -28.374, 112.036, -16.824, -83.07, 51.059]
  Set speed (120.0 mm/s)
  MoveL 10554 to (504.36, 506.75, 19.3) mm, rotated rx 0 ry 90 rz 0 deg; joints [-12.537, -28.213, 111.046, -16.589, -82.266, 51.27]
  Set speed (1000.0 mm/s)
  MoveL 10555 to (508.59, 493.75, 19.3) mm, rotated rx 0 ry 90 rz 0 deg; joints [-11.277, -28.183, 110.866, -15.324, -82.078, 51.157]
  Set speed (15.0 mm/s)
  Call Extruder(0.096)
  MoveL 10556 to (506.25, 491.4, 19.3) mm, rotated rx 0 ry 90 rz 0 deg; joints [-11.106, -28.24, 111.204, -15.141, -82.344, 51.062]
  Set speed (120.0 mm/s)
  MoveL 10557 to (507.24, 491.4, 19.3) mm, rotated rx 0 ry 90 rz 0 deg; joints [-11.088, -28.22, 111.085, -15.127, -82.247, 51.086]
  Set speed (15.0 mm/s)
  Call Extruder(0.056)
  MoveL 10558 to (508.59, 492.76, 19.3) mm, rotated rx 0 ry 90 rz 0 deg; joints [-11.187, -28.187, 110.89, -15.232, -82.094, 51.141]
  Set speed (120.0 mm/s)
  MoveL 10559 to (508.59, 491.76, 19.3) mm, rotated rx 0 ry 90 rz 0 deg; joints [-11.097, -28.191, 110.913, -15.141, -82.11, 51.124]
  Set speed (15.0 mm/s)
  Call Extruder(0.015)
  MoveL 10560 to (508.23, 491.4, 19.3) mm, rotated rx 0 ry 90 rz 0 deg; joints [-11.07, -28.2, 110.965, -15.112, -82.151, 51.11]
  Set speed (120.0 mm/s)
  MoveL 10561 to (495.89, 493.58, 19.3) mm, rotated rx 0 ry 90 rz 0 deg; joints [-11.496, -28.429, 112.393, -15.501, -83.32, 50.839]
  Set speed (1000.0 mm/s)
  MoveL 10562 to (490.47, 509.53, 19.3) mm, rotated rx 0 ry 90 rz 0 deg; joints [-13.08, -28.464, 112.624, -17.088, -83.554, 50.942]
  Set speed (1000.0 mm/s)
  MoveL 10563 to (490.4, 509.6, 19.3) mm, rotated rx 0 ry 90 rz 0 deg; joints [-13.088, -28.465, 112.63, -17.096, -83.559, 50.941]
  Set speed (1000.0 mm/s)
  MoveL 10564 to (490.4, 509.6, 19.4) mm, rotated rx 0 ry 90 rz 0 deg; joints [-13.088, -28.476, 112.635, -17.096, -83.554, 50.942]
  Set speed (15.0 mm/s)
  Call Extruder(0.559)
  MoveL 10565 to (490.4, 490.4, 19.4) mm, rotated rx 0 ry 90 rz 0 deg; joints [-11.303, -28.548, 113.126, -15.289, -83.907, 50.656]
  MoveL 10566 to (509.6, 490.4, 19.4) mm, rotated rx 0 ry 90 rz 0 deg; joints [-10.955, -28.186, 110.829, -15, -82.028, 51.128]
  MoveL 10567 to (509.6, 509.6, 19.4) mm, rotated rx 0 ry 90 rz 0 deg; joints [-12.688, -28.103, 110.344, -16.766, -81.704, 51.46]
  MoveL 10568 to (490.4, 509.6, 19.4) mm, rotated rx 0 ry 90 rz 0 deg; joints [-13.088, -28.476, 112.635, -17.096, -83.554, 50.942]
  Set speed (120.0 mm/s)
  MoveL 10569 to (490.4, 509.2, 19.4) mm, rotated rx 0 ry 90 rz 0 deg; joints [-13.051, -28.477, 112.646, -17.059, -83.562, 50.936]
  Set speed (1000.0 mm/s)
  MoveL 10570 to (490.5, 509.2, 19.4) mm, rotated rx 0 ry 90 rz 0 deg; joints [-13.049, -28.475, 112.635, -17.057, -83.552, 50.939]
  Set speed (1000.0 mm/s)
  MoveL 10571 to (495.94, 504.34, 19.4) mm, rotated rx 0 ry 90 rz 0 deg; joints [-12.487, -28.397, 112.121, -16.507, -83.118, 51.008]
  Set speed (1000.0 mm/s)
  MoveL 10572 to (496.01, 504.41, 19.4) mm, rotated rx 0 ry 90 rz 0 deg; joints [-12.492, -28.395, 112.111, -16.512, -83.11, 51.011]
  Set speed (15.0 mm/s)
  Call Extruder(0.067)
  MoveL 10573 to (496.01, 506.72, 19.4) mm, rotated rx 0 ry 90 rz 0 deg; joints [-12.705, -28.385, 112.049, -16.728, -83.067, 51.049]
  Call Extruder(0.242)
  MoveL 10574 to (504.33, 506.72, 19.4) mm, rotated rx 0 ry 90 rz 0 deg; joints [-12.535, -28.224, 111.055, -16.587, -82.264, 51.27]
  Call Extruder(0.027)
  MoveL 10575 to (504.33, 505.8, 19.4) mm, rotated rx 0 ry 90 rz 0 deg; joints [-12.452, -28.229, 111.08, -16.503, -82.28, 51.254]
  Call Extruder(0.306)
  MoveL 10576 to (499.53, 496.43, 19.4) mm, rotated rx 0 ry 90 rz 0 deg; joints [-11.69, -28.361, 111.894, -15.71, -82.91, 50.976]
  Call Extruder(0.017)
  MoveL 10577 to (499.27, 495.92, 19.4) mm, rotated rx 0 ry 90 rz 0 deg; joints [-11.648, -28.368, 111.938, -15.667, -82.945, 50.961]
  Call Extruder(0.010)
  MoveL 10578 to (499.84, 495.92, 19.4) mm, rotated rx 0 ry 90 rz 0 deg; joints [-11.637, -28.357, 111.87, -15.658, -82.889, 50.976]
  Call Extruder(0.000)
  MoveL 10579 to (499.84, 495.92, 19.4) mm, rotated rx 0 ry 90 rz 0 deg; joints [-11.637, -28.357, 111.869, -15.658, -82.889, 50.976]
  Call Extruder(0.136)
  MoveL 10580 to (504.51, 495.92, 19.4) mm, rotated rx 0 ry 90 rz 0 deg; joints [-11.55, -28.267, 111.31, -15.586, -82.434, 51.093]
  Call Extruder(0.067)
  MoveL 10581 to (504.51, 493.61, 19.4) mm, rotated rx 0 ry 90 rz 0 deg; joints [-11.338, -28.276, 111.366, -15.371, -82.473, 51.056]
  Call Extruder(0.250)
  MoveL 10582 to (495.92, 493.61, 19.4) mm, rotated rx 0 ry 90 rz 0 deg; joints [-11.498, -28.439, 112.394, -15.503, -83.311, 50.841]
  Call Extruder(0.027)
  MoveL 10583 to (495.92, 494.52, 19.4) mm, rotated rx 0 ry 90 rz 0 deg; joints [-11.583, -28.435, 112.371, -15.589, -83.295, 50.855]
  Call Extruder(0.306)
  MoveL 10584 to (500.7, 503.9, 19.4) mm, rotated rx 0 ry 90 rz 0 deg; joints [-12.351, -28.308, 111.564, -16.386, -82.665, 51.127]
  Call Extruder(0.017)
  MoveL 10585 to (500.96, 504.4, 19.4) mm, rotated rx 0 ry 90 rz 0 deg; joints [-12.392, -28.301, 111.52, -16.429, -82.631, 51.142]
  Call Extruder(0.010)
  MoveL 10586 to (500.39, 504.41, 19.4) mm, rotated rx 0 ry 90 rz 0 deg; joints [-12.404, -28.312, 111.588, -16.438, -82.686, 51.127]
  Call Extruder(0.000)
  MoveL 10587 to (500.39, 504.4, 19.4) mm, rotated rx 0 ry 90 rz 0 deg; joints [-12.404, -28.312, 111.588, -16.438, -82.686, 51.127]
  Call Extruder(0.128)
  MoveL 10588 to (496.01, 504.41, 19.4) mm, rotated rx 0 ry 90 rz 0 deg; joints [-12.492, -28.395, 112.111, -16.512, -83.11, 51.011]
  Set speed (120.0 mm/s)
  MoveL 10589 to (496.01, 504.81, 19.4) mm, rotated rx 0 ry 90 rz 0 deg; joints [-12.529, -28.393, 112.1, -16.549, -83.103, 51.017]
  Set speed (1000.0 mm/s)
  MoveL 10590 to (495.91, 504.81, 19.4) mm, rotated rx 0 ry 90 rz 0 deg; joints [-12.531, -28.395, 112.112, -16.551, -83.113, 51.015]
  Set speed (1000.0 mm/s)
  MoveL 10591 to (495.32, 503.72, 19.4) mm, rotated rx 0 ry 90 rz 0 deg; joints [-12.443, -28.411, 112.211, -16.459, -83.19, 50.982]
  Set speed (15.0 mm/s)
  Call Extruder(0.107)
  MoveL 10592 to (495.32, 507.41, 19.4) mm, rotated rx 0 ry 90 rz 0 deg; joints [-12.782, -28.395, 112.113, -16.804, -83.121, 51.041]
  Call Extruder(0.282)
  MoveL 10593 to (505.02, 507.41, 19.4) mm, rotated rx 0 ry 90 rz 0 deg; joints [-12.583, -28.207, 110.954, -16.639, -82.185, 51.3]
  Call Extruder(0.052)
  MoveL 10594 to (505.02, 505.64, 19.4) mm, rotated rx 0 ry 90 rz 0 deg; joints [-12.423, -28.215, 111.001, -16.476, -82.217, 51.269]
  Call Extruder(0.295)
  MoveL 10595 to (500.4, 496.61, 19.4) mm, rotated rx 0 ry 90 rz 0 deg; joints [-11.69, -28.344, 111.786, -15.714, -82.823, 51.001]
  Call Extruder(0.140)
  MoveL 10596 to (505.2, 496.61, 19.4) mm, rotated rx 0 ry 90 rz 0 deg; joints [-11.6, -28.25, 111.21, -15.639, -82.355, 51.122]
  Call Extruder(0.107)
  MoveL 10597 to (505.2, 492.92, 19.4) mm, rotated rx 0 ry 90 rz 0 deg; joints [-11.263, -28.265, 111.3, -15.297, -82.417, 51.062]
  Call Extruder(0.290)
  MoveL 10598 to (495.23, 492.92, 19.4) mm, rotated rx 0 ry 90 rz 0 deg; joints [-11.447, -28.454, 112.493, -15.449, -83.39, 50.814]
  Call Extruder(0.052)
  MoveL 10599 to (495.23, 494.69, 19.4) mm, rotated rx 0 ry 90 rz 0 deg; joints [-11.611, -28.447, 112.45, -15.616, -83.36, 50.84]
  Call Extruder(0.295)
  MoveL 10600 to (499.84, 503.72, 19.4) mm, rotated rx 0 ry 90 rz 0 deg; joints [-12.352, -28.326, 111.672, -16.383, -82.752, 51.101]
  Call Extruder(0.132)
  MoveL 10601 to (495.32, 503.72, 19.4) mm, rotated rx 0 ry 90 rz 0 deg; joints [-12.443, -28.411, 112.211, -16.459, -83.19, 50.982]
  Set speed (120.0 mm/s)
  MoveL 10602 to (491.09, 508.91, 19.4) mm, rotated rx 0 ry 90 rz 0 deg; joints [-13.01, -28.466, 112.573, -17.019, -83.501, 50.95]
  Set speed (15.0 mm/s)
  Call Extruder(0.519)
  MoveL 10603 to (491.09, 491.09, 19.4) mm, rotated rx 0 ry 90 rz 0 deg; joints [-11.355, -28.534, 113.028, -15.343, -83.827, 50.683]
  MoveL 10604 to (508.91, 491.09, 19.4) mm, rotated rx 0 ry 90 rz 0 deg; joints [-11.03, -28.198, 110.896, -15.074, -82.085, 51.122]
  MoveL 10605 to (508.91, 508.91, 19.4) mm, rotated rx 0 ry 90 rz 0 deg; joints [-12.64, -28.121, 110.445, -16.714, -81.783, 51.43]
  MoveL 10606 to (491.09, 508.91, 19.4) mm, rotated rx 0 ry 90 rz 0 deg; joints [-13.01, -28.466, 112.573, -17.019, -83.501, 50.95]
  Set speed (120.0 mm/s)
  MoveL 10607 to (491.4, 491.62, 19.4) mm, rotated rx 0 ry 90 rz 0 deg; joints [-11.398, -28.527, 112.979, -15.388, -83.787, 50.698]
  Set speed (15.0 mm/s)
  Call Extruder(0.009)
  MoveL 10608 to (491.61, 491.4, 19.4) mm, rotated rx 0 ry 90 rz 0 deg; joints [-11.374, -28.524, 112.959, -15.364, -83.77, 50.701]
  Set speed (120.0 mm/s)
  MoveL 10609 to (492.61, 491.4, 19.4) mm, rotated rx 0 ry 90 rz 0 deg; joints [-11.356, -28.506, 112.841, -15.349, -83.673, 50.725]
  Set speed (15.0 mm/s)
  Call Extruder(0.049)
  MoveL 10610 to (491.4, 492.61, 19.4) mm, rotated rx 0 ry 90 rz 0 deg; joints [-11.49, -28.523, 112.955, -15.481, -83.77, 50.712]
  Set speed (120.0 mm/s)
  MoveL 10611 to (491.4, 493.6, 19.4) mm, rotated rx 0 ry 90 rz 0 deg; joints [-11.583, -28.52, 112.931, -15.575, -83.753, 50.726]
  Set speed (15.0 mm/s)
  Call Extruder(0.090)
  MoveL 10612 to (493.6, 491.4, 19.4) mm, rotated rx 0 ry 90 rz 0 deg; joints [-11.337, -28.489, 112.723, -15.333, -83.576, 50.75]
  Set speed (120.0 mm/s)
  MoveL 10613 to (494.58, 491.4, 19.4) mm, rotated rx 0 ry 90 rz 0 deg; joints [-11.319, -28.471, 112.606, -15.317, -83.479, 50.775]
  Set speed (15.0 mm/s)
  Call Extruder(0.131)
  MoveL 10614 to (491.4, 494.58, 19.4) mm, rotated rx 0 ry 90 rz 0 deg; joints [-11.675, -28.516, 112.907, -15.668, -83.736, 50.741]
  Set speed (120.0 mm/s)
  MoveL 10615 to (491.4, 495.57, 19.4) mm, rotated rx 0 ry 90 rz 0 deg; joints [-11.767, -28.512, 112.882, -15.761, -83.718, 50.755]
  Set speed (15.0 mm/s)
  Call Extruder(0.172)
  MoveL 10616 to (495.57, 491.4, 19.4) mm, rotated rx 0 ry 90 rz 0 deg; joints [-11.3, -28.453, 112.488, -15.302, -83.382, 50.8]
  Set speed (120.0 mm/s)
  MoveL 10617 to (496.57, 491.4, 19.4) mm, rotated rx 0 ry 90 rz 0 deg; joints [-11.282, -28.435, 112.37, -15.287, -83.286, 50.824]
  Set speed (15.0 mm/s)
  Call Extruder(0.049)
  MoveL 10618 to (495.37, 492.6, 19.4) mm, rotated rx 0 ry 90 rz 0 deg; joints [-11.415, -28.453, 112.484, -15.418, -83.382, 50.812]
  Set speed (120.0 mm/s)
  MoveL 10619 to (494.92, 493.05, 19.4) mm, rotated rx 0 ry 90 rz 0 deg; joints [-11.466, -28.459, 112.527, -15.467, -83.419, 50.808]
  Set speed (15.0 mm/s)
  Call Extruder(0.145)
  MoveL 10620 to (491.4, 496.57, 19.4) mm, rotated rx 0 ry 90 rz 0 deg; joints [-11.859, -28.509, 112.858, -15.855, -83.7, 50.77]
  Set speed (120.0 mm/s)
  MoveL 10621 to (491.4, 497.55, 19.4) mm, rotated rx 0 ry 90 rz 0 deg; joints [-11.951, -28.505, 112.833, -15.948, -83.683, 50.784]
  Set speed (15.0 mm/s)
  Call Extruder(0.145)
  MoveL 10622 to (494.92, 494.04, 19.4) mm, rotated rx 0 ry 90 rz 0 deg; joints [-11.557, -28.456, 112.503, -15.56, -83.402, 50.822]
  Set speed (120.0 mm/s)
  MoveL 10623 to (495.01, 494.94, 19.4) mm, rotated rx 0 ry 90 rz 0 deg; joints [-11.639, -28.451, 112.47, -15.643, -83.377, 50.838]
  Set speed (15.0 mm/s)
  Call Extruder(0.148)
  MoveL 10624 to (491.4, 498.54, 19.4) mm, rotated rx 0 ry 90 rz 0 deg; joints [-12.043, -28.501, 112.808, -16.041, -83.665, 50.799]
  Set speed (120.0 mm/s)
  MoveL 10625 to (491.4, 499.53, 19.4) mm, rotated rx 0 ry 90 rz 0 deg; joints [-12.135, -28.498, 112.783, -16.134, -83.647, 50.814]
  Set speed (15.0 mm/s)
  Call Extruder(0.162)
  MoveL 10626 to (495.34, 495.6, 19.4) mm, rotated rx 0 ry 90 rz 0 deg; joints [-11.693, -28.442, 112.414, -15.699, -83.333, 50.856]
  Set speed (120.0 mm/s)
  MoveL 10627 to (495.68, 496.25, 19.4) mm, rotated rx 0 ry 90 rz 0 deg; joints [-11.747, -28.433, 112.358, -15.755, -83.289, 50.875]
  Set speed (15.0 mm/s)
  Call Extruder(0.176)
  MoveL 10628 to (491.4, 500.52, 19.4) mm, rotated rx 0 ry 90 rz 0 deg; joints [-12.227, -28.494, 112.758, -16.227, -83.629, 50.829]
  Set speed (120.0 mm/s)
  MoveL 10629 to (491.4, 501.51, 19.4) mm, rotated rx 0 ry 90 rz 0 deg; joints [-12.319, -28.49, 112.732, -16.32, -83.61, 50.844]
  Set speed (15.0 mm/s)
  Call Extruder(0.190)
  MoveL 10630 to (496.01, 496.91, 19.4) mm, rotated rx 0 ry 90 rz 0 deg; joints [-11.802, -28.425, 112.302, -15.811, -83.245, 50.893]
  Set speed (120.0 mm/s)
  MoveL 10631 to (496.34, 497.56, 19.4) mm, rotated rx 0 ry 90 rz 0 deg; joints [-11.856, -28.416, 112.246, -15.867, -83.201, 50.912]
  Set speed (15.0 mm/s)
  Call Extruder(0.203)
  MoveL 10632 to (491.4, 502.5, 19.4) mm, rotated rx 0 ry 90 rz 0 deg; joints [-12.411, -28.486, 112.707, -16.413, -83.592, 50.859]
  Set speed (120.0 mm/s)
  MoveL 10633 to (491.4, 503.49, 19.4) mm, rotated rx 0 ry 90 rz 0 deg; joints [-12.502, -28.482, 112.681, -16.506, -83.574, 50.874]
  Set speed (15.0 mm/s)
  Call Extruder(0.217)
  MoveL 10634 to (496.68, 498.22, 19.4) mm, rotated rx 0 ry 90 rz 0 deg; joints [-11.91, -28.407, 112.19, -15.923, -83.157, 50.931]
  Set speed (120.0 mm/s)
  MoveL 10635 to (497.01, 498.88, 19.4) mm, rotated rx 0 ry 90 rz 0 deg; joints [-11.964, -28.399, 112.134, -15.979, -83.113, 50.95]
  Set speed (15.0 mm/s)
  Call Extruder(0.231)
  MoveL 10636 to (491.4, 504.48, 19.4) mm, rotated rx 0 ry 90 rz 0 deg; joints [-12.594, -28.478, 112.655, -16.599, -83.555, 50.889]
  Set speed (120.0 mm/s)
  MoveL 10637 to (491.4, 505.47, 19.4) mm, rotated rx 0 ry 90 rz 0 deg; joints [-12.686, -28.474, 112.628, -16.692, -83.536, 50.905]
  Set speed (15.0 mm/s)
  Call Extruder(0.245)
  MoveL 10638 to (497.35, 499.53, 19.4) mm, rotated rx 0 ry 90 rz 0 deg; joints [-12.017, -28.39, 112.077, -16.035, -83.069, 50.969]
  Set speed (120.0 mm/s)
  MoveL 10639 to (497.68, 500.19, 19.4) mm, rotated rx 0 ry 90 rz 0 deg; joints [-12.071, -28.381, 112.021, -16.091, -83.024, 50.988]
  Set speed (15.0 mm/s)
  Call Extruder(0.258)
  MoveL 10640 to (491.4, 506.46, 19.4) mm, rotated rx 0 ry 90 rz 0 deg; joints [-12.777, -28.47, 112.602, -16.785, -83.517, 50.92]
  Set speed (120.0 mm/s)
  MoveL 10641 to (491.4, 507.45, 19.4) mm, rotated rx 0 ry 90 rz 0 deg; joints [-12.868, -28.466, 112.575, -16.877, -83.498, 50.936]
  Set speed (15.0 mm/s)
  Call Extruder(0.148)
  MoveL 10642 to (495, 503.86, 19.4) mm, rotated rx 0 ry 90 rz 0 deg; joints [-12.462, -28.416, 112.245, -16.478, -83.218, 50.976]
  Set speed (120.0 mm/s)
  MoveL 10643 to (495.46, 503.4, 19.4) mm, rotated rx 0 ry 90 rz 0 deg; joints [-12.411, -28.409, 112.202, -16.427, -83.182, 50.98]
  Set speed (15.0 mm/s)
  Call Extruder(0.105)
  MoveL 10644 to (498.02, 500.84, 19.4) mm, rotated rx 0 ry 90 rz 0 deg; joints [-12.125, -28.372, 111.964, -16.146, -82.98, 51.007]
  Set speed (120.0 mm/s)
  MoveL 10645 to (498.35, 501.5, 19.4) mm, rotated rx 0 ry 90 rz 0 deg; joints [-12.178, -28.363, 111.907, -16.202, -82.936, 51.026]
  Set speed (15.0 mm/s)
  Call Extruder(0.078)
  MoveL 10646 to (496.45, 503.4, 19.4) mm, rotated rx 0 ry 90 rz 0 deg; joints [-12.391, -28.391, 112.084, -16.411, -83.086, 51.007]
  Set speed (120.0 mm/s)
  MoveL 10647 to (497.44, 503.4, 19.4) mm, rotated rx 0 ry 90 rz 0 deg; joints [-12.371, -28.372, 111.966, -16.394, -82.99, 51.033]
  Set speed (15.0 mm/s)
  Call Extruder(0.051)
  MoveL 10648 to (498.68, 502.15, 19.4) mm, rotated rx 0 ry 90 rz 0 deg; joints [-12.232, -28.354, 111.85, -16.257, -82.892, 51.045]
  Set speed (120.0 mm/s)
  MoveL 10649 to (499.02, 502.81, 19.4) mm, rotated rx 0 ry 90 rz 0 deg; joints [-12.285, -28.345, 111.793, -16.313, -82.848, 51.065]
  Set speed (15.0 mm/s)
  Call Extruder(0.024)
  MoveL 10650 to (498.43, 503.4, 19.4) mm, rotated rx 0 ry 90 rz 0 deg; joints [-12.351, -28.354, 111.848, -16.377, -82.894, 51.059]
  Set speed (120.0 mm/s)
  MoveL 10651 to (496.45, 504.19, 19.4) mm, rotated rx 0 ry 90 rz 0 deg; joints [-12.464, -28.388, 112.064, -16.485, -83.072, 51.019]
  Set speed (1000.0 mm/s)
  MoveL 10652 to (495, 504.85, 19.4) mm, rotated rx 0 ry 90 rz 0 deg; joints [-12.554, -28.412, 112.219, -16.57, -83.2, 50.991]
  Set speed (15.0 mm/s)
  Call Extruder(0.148)
  MoveL 10653 to (491.4, 508.44, 19.4) mm, rotated rx 0 ry 90 rz 0 deg; joints [-12.96, -28.462, 112.548, -16.97, -83.479, 50.952]
  Set speed (120.0 mm/s)
  MoveL 10654 to (492.24, 508.59, 19.4) mm, rotated rx 0 ry 90 rz 0 deg; joints [-12.956, -28.447, 112.445, -16.969, -83.395, 50.977]
  Set speed (15.0 mm/s)
  Call Extruder(0.113)
  MoveL 10655 to (495, 505.84, 19.4) mm, rotated rx 0 ry 90 rz 0 deg; joints [-12.645, -28.408, 112.192, -16.663, -83.181, 51.007]
  Set speed (120.0 mm/s)
  MoveL 10656 to (495, 506.83, 19.4) mm, rotated rx 0 ry 90 rz 0 deg; joints [-12.735, -28.404, 112.166, -16.755, -83.163, 51.023]
  Set speed (15.0 mm/s)
  Call Extruder(0.073)
  MoveL 10657 to (493.23, 508.59, 19.4) mm, rotated rx 0 ry 90 rz 0 deg; joints [-12.935, -28.429, 112.328, -16.951, -83.3, 51.004]
  Set speed (120.0 mm/s)
  MoveL 10658 to (494.22, 508.59, 19.4) mm, rotated rx 0 ry 90 rz 0 deg; joints [-12.914, -28.411, 112.21, -16.934, -83.204, 51.031]
  Set speed (15.0 mm/s)
  Call Extruder(0.036)
  MoveL 10659 to (495.1, 507.72, 19.4) mm, rotated rx 0 ry 90 rz 0 deg; joints [-12.816, -28.398, 112.13, -16.837, -83.136, 51.04]
  Set speed (120.0 mm/s)
  MoveL 10660 to (495.21, 508.59, 19.4) mm, rotated rx 0 ry 90 rz 0 deg; joints [-12.893, -28.392, 112.093, -16.916, -83.108, 51.058]
  Set speed (15.0 mm/s)
  MoveL 10661 to (496.09, 507.72, 19.4) mm, rotated rx 0 ry 90 rz 0 deg; joints [-12.795, -28.38, 112.013, -16.819, -83.041, 51.067]
  Set speed (120.0 mm/s)
  MoveL 10662 to (496.2, 508.59, 19.4) mm, rotated rx 0 ry 90 rz 0 deg; joints [-12.872, -28.374, 111.975, -16.899, -83.013, 51.085]
  Set speed (15.0 mm/s)
  Call Extruder(0.036)
  MoveL 10663 to (497.08, 507.72, 19.4) mm, rotated rx 0 ry 90 rz 0 deg; joints [-12.774, -28.361, 111.895, -16.802, -82.945, 51.094]
  Set speed (120.0 mm/s)
  MoveL 10664 to (497.19, 508.59, 19.4) mm, rotated rx 0 ry 90 rz 0 deg; joints [-12.852, -28.355, 111.857, -16.881, -82.917, 51.111]
  Set speed (15.0 mm/s)
  MoveL 10665 to (498.07, 507.72, 19.4) mm, rotated rx 0 ry 90 rz 0 deg; joints [-12.754, -28.342, 111.777, -16.785, -82.85, 51.12]
  Set speed (120.0 mm/s)
  MoveL 10666 to (498.18, 508.59, 19.4) mm, rotated rx 0 ry 90 rz 0 deg; joints [-12.831, -28.336, 111.739, -16.864, -82.822, 51.138]
  Set speed (15.0 mm/s)
  MoveL 10667 to (499.06, 507.72, 19.4) mm, rotated rx 0 ry 90 rz 0 deg; joints [-12.733, -28.323, 111.659, -16.768, -82.754, 51.147]
  Set speed (120.0 mm/s)
  MoveL 10668 to (499.17, 508.59, 19.4) mm, rotated rx 0 ry 90 rz 0 deg; joints [-12.811, -28.317, 111.621, -16.847, -82.726, 51.165]
  Set speed (15.0 mm/s)
  MoveL 10669 to (500.05, 507.72, 19.4) mm, rotated rx 0 ry 90 rz 0 deg; joints [-12.713, -28.304, 111.541, -16.751, -82.658, 51.173]
  Set speed (120.0 mm/s)
  MoveL 10670 to (500.16, 508.59, 19.4) mm, rotated rx 0 ry 90 rz 0 deg; joints [-12.79, -28.298, 111.503, -16.83, -82.631, 51.191]
  Set speed (15.0 mm/s)
  MoveL 10671 to (501.04, 507.72, 19.4) mm, rotated rx 0 ry 90 rz 0 deg; joints [-12.693, -28.285, 111.423, -16.735, -82.563, 51.2]
  Set speed (120.0 mm/s)
  MoveL 10672 to (501.15, 508.59, 19.4) mm, rotated rx 0 ry 90 rz 0 deg; joints [-12.77, -28.279, 111.385, -16.813, -82.535, 51.218]
  Set speed (15.0 mm/s)
  MoveL 10673 to (502.03, 507.72, 19.4) mm, rotated rx 0 ry 90 rz 0 deg; joints [-12.672, -28.266, 111.304, -16.718, -82.467, 51.226]
  Set speed (120.0 mm/s)
  MoveL 10674 to (502.14, 508.59, 19.4) mm, rotated rx 0 ry 90 rz 0 deg; joints [-12.749, -28.26, 111.267, -16.797, -82.44, 51.244]
  Set speed (15.0 mm/s)
  MoveL 10675 to (503.02, 507.72, 19.4) mm, rotated rx 0 ry 90 rz 0 deg; joints [-12.652, -28.246, 111.186, -16.701, -82.372, 51.253]
  Set speed (120.0 mm/s)
  MoveL 10676 to (503.13, 508.59, 19.4) mm, rotated rx 0 ry 90 rz 0 deg; joints [-12.729, -28.24, 111.148, -16.78, -82.345, 51.271]
  Set speed (15.0 mm/s)
  MoveL 10677 to (504.01, 507.72, 19.4) mm, rotated rx 0 ry 90 rz 0 deg; joints [-12.632, -28.226, 111.067, -16.685, -82.277, 51.279]
  Set speed (120.0 mm/s)
  MoveL 10678 to (504.12, 508.59, 19.4) mm, rotated rx 0 ry 90 rz 0 deg; joints [-12.709, -28.22, 111.029, -16.763, -82.249, 51.297]
  Set speed (15.0 mm/s)
  MoveL 10679 to (505, 507.72, 19.4) mm, rotated rx 0 ry 90 rz 0 deg; joints [-12.612, -28.207, 110.948, -16.669, -82.181, 51.305]
  Set speed (120.0 mm/s)
  MoveL 10680 to (505.33, 507.39, 19.4) mm, rotated rx 0 ry 90 rz 0 deg; joints [-12.575, -28.201, 110.917, -16.632, -82.155, 51.308]
  Set speed (15.0 mm/s)
  Call Extruder(0.134)
  MoveL 10681 to (508.59, 504.12, 19.4) mm, rotated rx 0 ry 90 rz 0 deg; joints [-12.216, -28.149, 110.611, -16.28, -81.898, 51.336]
  Set speed (120.0 mm/s)
  MoveL 10682 to (508.59, 505.11, 19.4) mm, rotated rx 0 ry 90 rz 0 deg; joints [-12.305, -28.145, 110.585, -16.371, -81.881, 51.353]
  Set speed (15.0 mm/s)
  Call Extruder(0.143)
  MoveL 10683 to (505.11, 508.59, 19.4) mm, rotated rx 0 ry 90 rz 0 deg; joints [-12.689, -28.2, 110.911, -16.747, -82.154, 51.323]
  Set speed (120.0 mm/s)
  MoveL 10684 to (506.1, 508.59, 19.4) mm, rotated rx 0 ry 90 rz 0 deg; joints [-12.668, -28.18, 110.792, -16.731, -82.059, 51.35]
  Set speed (15.0 mm/s)
  Call Extruder(0.103)
  MoveL 10685 to (508.59, 506.1, 19.4) mm, rotated rx 0 ry 90 rz 0 deg; joints [-12.394, -28.14, 110.559, -16.461, -81.863, 51.371]
  Set speed (120.0 mm/s)
  MoveL 10686 to (508.59, 507.09, 19.4) mm, rotated rx 0 ry 90 rz 0 deg; joints [-12.483, -28.136, 110.532, -16.552, -81.846, 51.389]
  Set speed (15.0 mm/s)
  Call Extruder(0.062)
  MoveL 10687 to (507.09, 508.59, 19.4) mm, rotated rx 0 ry 90 rz 0 deg; joints [-12.648, -28.16, 110.673, -16.714, -81.963, 51.376]
  Set speed (120.0 mm/s)
  MoveL 10688 to (508.08, 508.59, 19.4) mm, rotated rx 0 ry 90 rz 0 deg; joints [-12.628, -28.139, 110.554, -16.698, -81.868, 51.402]
  Set speed (15.0 mm/s)
  Call Extruder(0.021)
  MoveL 10689 to (508.59, 508.08, 19.4) mm, rotated rx 0 ry 90 rz 0 deg; joints [-12.572, -28.131, 110.506, -16.643, -81.828, 51.406]
  Set speed (120.0 mm/s)
  MoveL 10690 to (505.33, 506.4, 19.4) mm, rotated rx 0 ry 90 rz 0 deg; joints [-12.485, -28.206, 110.943, -16.541, -82.173, 51.291]
  Set speed (15.0 mm/s)
  Call Extruder(0.134)
  MoveL 10691 to (508.59, 503.13, 19.4) mm, rotated rx 0 ry 90 rz 0 deg; joints [-12.126, -28.154, 110.636, -16.189, -81.915, 51.319]
  Set speed (120.0 mm/s)
  MoveL 10692 to (508.59, 502.14, 19.4) mm, rotated rx 0 ry 90 rz 0 deg; joints [-12.037, -28.158, 110.662, -16.098, -81.932, 51.301]
  Set speed (15.0 mm/s)
  Call Extruder(0.136)
  MoveL 10693 to (505.28, 505.46, 19.4) mm, rotated rx 0 ry 90 rz 0 deg; joints [-12.402, -28.211, 110.974, -16.455, -82.194, 51.273]
  Set speed (120.0 mm/s)
  MoveL 10694 to (504.94, 504.8, 19.4) mm, rotated rx 0 ry 90 rz 0 deg; joints [-12.349, -28.221, 111.032, -16.4, -82.239, 51.253]
  Set speed (15.0 mm/s)
  Call Extruder(0.150)
  MoveL 10695 to (508.59, 501.15, 19.4) mm, rotated rx 0 ry 90 rz 0 deg; joints [-11.948, -28.162, 110.687, -16.007, -81.949, 51.284]
  Set speed (120.0 mm/s)
  MoveL 10696 to (508.59, 500.16, 19.4) mm, rotated rx 0 ry 90 rz 0 deg; joints [-11.858, -28.167, 110.712, -15.916, -81.966, 51.267]
  Set speed (15.0 mm/s)
  Call Extruder(0.164)
  MoveL 10697 to (504.61, 504.15, 19.4) mm, rotated rx 0 ry 90 rz 0 deg; joints [-12.296, -28.23, 111.089, -16.345, -82.283, 51.233]
  Set speed (120.0 mm/s)
  MoveL 10698 to (504.27, 503.49, 19.4) mm, rotated rx 0 ry 90 rz 0 deg; joints [-12.243, -28.24, 111.147, -16.29, -82.327, 51.213]
  Set speed (15.0 mm/s)
  Call Extruder(0.178)
  MoveL 10699 to (508.59, 499.17, 19.4) mm, rotated rx 0 ry 90 rz 0 deg; joints [-11.769, -28.171, 110.737, -15.824, -81.983, 51.25]
  Set speed (120.0 mm/s)
  MoveL 10700 to (508.59, 498.18, 19.4) mm, rotated rx 0 ry 90 rz 0 deg; joints [-11.679, -28.175, 110.762, -15.733, -81.999, 51.233]
  Set speed (15.0 mm/s)
  Call Extruder(0.192)
  MoveL 10701 to (503.94, 502.84, 19.4) mm, rotated rx 0 ry 90 rz 0 deg; joints [-12.191, -28.249, 111.204, -16.235, -82.371, 51.193]
  Set speed (120.0 mm/s)
  MoveL 10702 to (503.6, 502.18, 19.4) mm, rotated rx 0 ry 90 rz 0 deg; joints [-12.138, -28.259, 111.261, -16.18, -82.415, 51.174]
  Set speed (15.0 mm/s)
  Call Extruder(0.205)
  MoveL 10703 to (508.59, 497.19, 19.4) mm, rotated rx 0 ry 90 rz 0 deg; joints [-11.589, -28.179, 110.787, -15.642, -82.016, 51.216]
  Set speed (120.0 mm/s)
  MoveL 10704 to (508.59, 496.2, 19.4) mm, rotated rx 0 ry 90 rz 0 deg; joints [-11.5, -28.183, 110.811, -15.551, -82.032, 51.2]
  Set speed (15.0 mm/s)
  Call Extruder(0.219)
  MoveL 10705 to (503.27, 501.53, 19.4) mm, rotated rx 0 ry 90 rz 0 deg; joints [-12.084, -28.268, 111.318, -16.125, -82.458, 51.154]
  Set speed (120.0 mm/s)
  MoveL 10706 to (502.93, 500.87, 19.4) mm, rotated rx 0 ry 90 rz 0 deg; joints [-12.031, -28.277, 111.375, -16.07, -82.503, 51.135]
  Set speed (15.0 mm/s)
  Call Extruder(0.233)
  MoveL 10707 to (508.59, 495.21, 19.4) mm, rotated rx 0 ry 90 rz 0 deg; joints [-11.41, -28.187, 110.835, -15.459, -82.049, 51.183]
  Set speed (120.0 mm/s)
  MoveL 10708 to (508.59, 494.22, 19.4) mm, rotated rx 0 ry 90 rz 0 deg; joints [-11.32, -28.192, 110.859, -15.368, -82.065, 51.166]
  Set speed (15.0 mm/s)
  Call Extruder(0.247)
  MoveL 10709 to (502.6, 500.22, 19.4) mm, rotated rx 0 ry 90 rz 0 deg; joints [-11.978, -28.287, 111.432, -16.014, -82.546, 51.115]
  Set speed (120.0 mm/s)
  MoveL 10710 to (502.26, 499.57, 19.4) mm, rotated rx 0 ry 90 rz 0 deg; joints [-11.925, -28.296, 111.489, -15.959, -82.59, 51.096]
  Set speed (15.0 mm/s)
  Call Extruder(0.109)
  MoveL 10711 to (504.9, 496.92, 19.4) mm, rotated rx 0 ry 90 rz 0 deg; joints [-11.634, -28.255, 111.238, -15.673, -82.379, 51.119]
  Set speed (120.0 mm/s)
  MoveL 10712 to (505.52, 496.31, 19.4) mm, rotated rx 0 ry 90 rz 0 deg; joints [-11.567, -28.245, 111.179, -15.607, -82.33, 51.125]
  Set speed (15.0 mm/s)
  Call Extruder(0.127)
  MoveL 10713 to (508.59, 493.23, 19.4) mm, rotated rx 0 ry 90 rz 0 deg; joints [-11.23, -28.196, 110.883, -15.277, -82.081, 51.15]
  Set speed (120.0 mm/s)
  MoveL 10714 to (508.59, 492.24, 19.4) mm, rotated rx 0 ry 90 rz 0 deg; joints [-11.14, -28.2, 110.907, -15.185, -82.097, 51.134]
  Set speed (15.0 mm/s)
  MoveL 10715 to (505.52, 495.32, 19.4) mm, rotated rx 0 ry 90 rz 0 deg; joints [-11.476, -28.249, 111.204, -15.515, -82.346, 51.108]
  Set speed (120.0 mm/s)
  MoveL 10716 to (505.52, 494.33, 19.4) mm, rotated rx 0 ry 90 rz 0 deg; joints [-11.386, -28.253, 111.228, -15.424, -82.363, 51.092]
  Set speed (15.0 mm/s)
  Call Extruder(0.121)
  MoveL 10717 to (508.44, 491.4, 19.4) mm, rotated rx 0 ry 90 rz 0 deg; joints [-11.067, -28.206, 110.945, -15.11, -82.125, 51.116]
  Set speed (120.0 mm/s)
  MoveL 10718 to (507.45, 491.4, 19.4) mm, rotated rx 0 ry 90 rz 0 deg; joints [-11.084, -28.226, 111.064, -15.124, -82.222, 51.092]
  Set speed (15.0 mm/s)
  Call Extruder(0.080)
  MoveL 10719 to (505.52, 493.34, 19.4) mm, rotated rx 0 ry 90 rz 0 deg; joints [-11.296, -28.257, 111.252, -15.332, -82.379, 51.076]
  Set speed (120.0 mm/s)
  MoveL 10720 to (505.27, 492.6, 19.4) mm, rotated rx 0 ry 90 rz 0 deg; joints [-11.233, -28.265, 111.299, -15.267, -82.416, 51.058]
  Set speed (15.0 mm/s)
  Call Extruder(0.049)
  MoveL 10721 to (506.46, 491.4, 19.4) mm, rotated rx 0 ry 90 rz 0 deg; joints [-11.102, -28.246, 111.184, -15.138, -82.318, 51.068]
  Set speed (120.0 mm/s)
  MoveL 10722 to (505.47, 491.4, 19.4) mm, rotated rx 0 ry 90 rz 0 deg; joints [-11.12, -28.266, 111.303, -15.153, -82.415, 51.044]
  Set speed (15.0 mm/s)
  MoveL 10723 to (504.28, 492.6, 19.4) mm, rotated rx 0 ry 90 rz 0 deg; joints [-11.251, -28.284, 111.418, -15.281, -82.512, 51.034]
  Set speed (120.0 mm/s)
  MoveL 10724 to (503.29, 492.6, 19.4) mm, rotated rx 0 ry 90 rz 0 deg; joints [-11.269, -28.304, 111.537, -15.296, -82.609, 51.009]
  Set speed (15.0 mm/s)
  MoveL 10725 to (504.48, 491.4, 19.4) mm, rotated rx 0 ry 90 rz 0 deg; joints [-11.137, -28.285, 111.422, -15.167, -82.511, 51.02]
  Set speed (120.0 mm/s)
  MoveL 10726 to (503.49, 491.4, 19.4) mm, rotated rx 0 ry 90 rz 0 deg; joints [-11.155, -28.304, 111.541, -15.182, -82.608, 50.996]
  Set speed (15.0 mm/s)
  MoveL 10727 to (502.3, 492.6, 19.4) mm, rotated rx 0 ry 90 rz 0 deg; joints [-11.287, -28.323, 111.656, -15.311, -82.705, 50.985]
  Set speed (120.0 mm/s)
  MoveL 10728 to (501.31, 492.6, 19.4) mm, rotated rx 0 ry 90 rz 0 deg; joints [-11.305, -28.342, 111.775, -15.326, -82.802, 50.96]
  Set speed (15.0 mm/s)
  MoveL 10729 to (502.5, 491.4, 19.4) mm, rotated rx 0 ry 90 rz 0 deg; joints [-11.173, -28.324, 111.66, -15.196, -82.705, 50.971]
  Set speed (120.0 mm/s)
  MoveL 10730 to (501.51, 491.4, 19.4) mm, rotated rx 0 ry 90 rz 0 deg; joints [-11.191, -28.343, 111.778, -15.211, -82.802, 50.947]
  Set speed (15.0 mm/s)
  MoveL 10731 to (500.32, 492.6, 19.4) mm, rotated rx 0 ry 90 rz 0 deg; joints [-11.323, -28.361, 111.893, -15.341, -82.899, 50.936]
  Set speed (120.0 mm/s)
  MoveL 10732 to (499.33, 492.6, 19.4) mm, rotated rx 0 ry 90 rz 0 deg; joints [-11.342, -28.38, 112.012, -15.356, -82.995, 50.911]
  Set speed (15.0 mm/s)
  MoveL 10733 to (500.52, 491.4, 19.4) mm, rotated rx 0 ry 90 rz 0 deg; joints [-11.209, -28.361, 111.897, -15.226, -82.898, 50.923]
  Set speed (120.0 mm/s)
  MoveL 10734 to (499.53, 491.4, 19.4) mm, rotated rx 0 ry 90 rz 0 deg; joints [-11.227, -28.38, 112.015, -15.241, -82.995, 50.898]
  Set speed (15.0 mm/s)
  Call Extruder(0.049)
  MoveL 10735 to (498.34, 492.6, 19.4) mm, rotated rx 0 ry 90 rz 0 deg; joints [-11.36, -28.398, 112.13, -15.371, -83.092, 50.887]
  Set speed (120.0 mm/s)
  MoveL 10736 to (497.35, 492.6, 19.4) mm, rotated rx 0 ry 90 rz 0 deg; joints [-11.378, -28.416, 112.248, -15.387, -83.189, 50.862]
  Set speed (15.0 mm/s)
  MoveL 10737 to (498.54, 491.4, 19.4) mm, rotated rx 0 ry 90 rz 0 deg; joints [-11.245, -28.399, 112.134, -15.256, -83.092, 50.874]
  Set speed (120.0 mm/s)
  MoveL 10738 to (497.55, 491.4, 19.4) mm, rotated rx 0 ry 90 rz 0 deg; joints [-11.264, -28.417, 112.252, -15.271, -83.189, 50.849]
  Set speed (15.0 mm/s)
  MoveL 10739 to (496.36, 492.6, 19.4) mm, rotated rx 0 ry 90 rz 0 deg; joints [-11.397, -28.435, 112.366, -15.402, -83.286, 50.837]
  MoveL 10740 to (496.23, 492.73, 19.4) mm, rotated rx 0 ry 90 rz 0 deg; joints [-11.41, -28.436, 112.378, -15.416, -83.296, 50.836]
  Set speed (120.0 mm/s)
  MoveL 10741 to (504.54, 493.58, 19.4) mm, rotated rx 0 ry 90 rz 0 deg; joints [-11.335, -28.275, 111.363, -15.368, -82.47, 51.056]
  Set speed (1000.0 mm/s)
  MoveL 10742 to (504.54, 495.95, 19.4) mm, rotated rx 0 ry 90 rz 0 deg; joints [-11.552, -28.266, 111.306, -15.588, -82.431, 51.094]
  Set speed (1000.0 mm/s)
  MoveL 10743 to (501.26, 497.6, 19.4) mm, rotated rx 0 ry 90 rz 0 deg; joints [-11.764, -28.323, 111.658, -15.792, -82.722, 51.038]
  Set speed (15.0 mm/s)
  Call Extruder(0.028)
  MoveL 10744 to (501.93, 496.92, 19.4) mm, rotated rx 0 ry 90 rz 0 deg; joints [-11.69, -28.313, 111.594, -15.719, -82.668, 51.045]
  Set speed (120.0 mm/s)
  MoveL 10745 to (502.92, 496.92, 19.4) mm, rotated rx 0 ry 90 rz 0 deg; joints [-11.671, -28.294, 111.476, -15.703, -82.572, 51.07]
  Set speed (15.0 mm/s)
  Call Extruder(0.055)
  MoveL 10746 to (501.59, 498.26, 19.4) mm, rotated rx 0 ry 90 rz 0 deg; joints [-11.818, -28.314, 111.602, -15.848, -82.678, 51.057]
  Set speed (120.0 mm/s)
  MoveL 10747 to (501.93, 498.91, 19.4) mm, rotated rx 0 ry 90 rz 0 deg; joints [-11.871, -28.305, 111.545, -15.903, -82.634, 51.077]
  Set speed (15.0 mm/s)
  Call Extruder(0.082)
  MoveL 10748 to (503.91, 496.92, 19.4) mm, rotated rx 0 ry 90 rz 0 deg; joints [-11.652, -28.274, 111.357, -15.688, -82.475, 51.094]
  MoveL 10749 to (504.04, 496.8, 19.4) mm, rotated rx 0 ry 90 rz 0 deg; joints [-11.639, -28.272, 111.345, -15.675, -82.466, 51.096]
  Set speed (120.0 mm/s)
  MoveL 10750 to (504.37, 505.79, 19.4) mm, rotated rx 0 ry 90 rz 0 deg; joints [-12.45, -28.228, 111.075, -16.501, -82.277, 51.255]
  Set speed (1000.0 mm/s)
  MoveL 10751 to (490.47, 509.53, 19.4) mm, rotated rx 0 ry 90 rz 0 deg; joints [-13.08, -28.475, 112.629, -17.089, -83.548, 50.943]
  Set speed (1000.0 mm/s)
  MoveL 10752 to (490.4, 509.6, 19.4) mm, rotated rx 0 ry 90 rz 0 deg; joints [-13.088, -28.476, 112.635, -17.096, -83.554, 50.942]
  Set speed (1000.0 mm/s)
  MoveL 10753 to (490.4, 509.6, 19.5) mm, rotated rx 0 ry 90 rz 0 deg; joints [-13.088, -28.486, 112.64, -17.097, -83.549, 50.944]
  Set speed (15.0 mm/s)
  Call Extruder(0.559)
  MoveL 10754 to (490.4, 490.4, 19.5) mm, rotated rx 0 ry 90 rz 0 deg; joints [-11.303, -28.559, 113.131, -15.289, -83.901, 50.657]
